(* PLC project pj23SH01.project, CODESYS CODESYS V3.5 SP18 Patch 2 *)
(* stored: creationDateTime 2023-05-12T09:11:09.1774968, modificationDateTime 2023-05-12T09:10:59.1943593 *)

TYPE EASY_object_manager_struct_t : STRUCT
  xFlip : BOOL;  (* commands *)
  xLoaded : BOOL;  (* feedbacks *)
  MarkerPose : ROS_pose_struct_t;
  xMarkerDetected : BOOL;
  xIsFlipped : BOOL;
  xResult_OK : BOOL;  (* elaboration *)
  xResult_NOT_OK : BOOL;
END_STRUCT;
END_TYPE

{attribute 'qualified_only'}
{attribute 'strict'}
TYPE piece_state_enum_t : (PieceUnknownState, PieceOK, PieceNotOK) UDINT;
END_TYPE

{attribute 'qualified_only'}
{attribute 'strict'}
TYPE manipulator_state_enum_t : (ManipulatorUnknownState, ManipulatorReady, ManipulatorRunning, ManipulatorError) UDINT;
END_TYPE

{attribute 'qualified_only'}
{attribute 'strict'}
TYPE piece_error_enum_t : (PIECE_NO_ERROR, PIECE_IN_WRONG_CONFIG, PIECE_NOT_FOUND) UDINT;
END_TYPE

{attribute 'qualified_only'}
{attribute 'strict'}
TYPE manipulator_error_enum_t : (MANIP_NO_ERROR, MANIP_GENERAL_ERROR, MANIP_EM_STOP, MANIP_EXEC_FAILED) UDINT;
END_TYPE

TYPE full_machine_struct_t : STRUCT
  Machine : machine_struct_t;
  Details : machine_details_struct_t;
  Counters : counters_interface_struct_t;
END_STRUCT;
END_TYPE

TYPE piece_struct_t : STRUCT
  xEnable : BOOL;
  eState : piece_state_enum_t;
  eError : piece_error_enum_t;
END_STRUCT;
END_TYPE

TYPE machine_struct_t : STRUCT
  xEnable : BOOL;
  eState : machine_state_enum_t;
  eError : machine_error_enum_t;
  sErrorMessage : STRING(255);
END_STRUCT;
END_TYPE

TYPE machine_details_struct_t : STRUCT
  aPieces : ARRAY[0..1] OF piece_struct_t;
  Manipulator : manipulator_struct_t;
END_STRUCT;
END_TYPE

TYPE manipulator_struct_t : STRUCT
  xEnable : BOOL;
  eState : manipulator_state_enum_t;
  eError : manipulator_error_enum_t;
END_STRUCT;
END_TYPE

TYPE counters_struct_t : STRUCT
  udiPiecesOK_Counter : UDINT;
  udiPiecesNotOK_Counter : UDINT;
  dtUTCStartCounting : DT;  (* time *)
  dwUpTime : DWORD;  (* in seconds *)
  dwReadyTime : DWORD;
  dwRunningTime : DWORD;  (* in seconds *)
  dwErrorTime : DWORD;  (* in seconds *)
END_STRUCT;
END_TYPE

TYPE counters_interface_struct_t : STRUCT
  LastSession : counters_struct_t;
  Overall : counters_struct_t;
END_STRUCT;
END_TYPE

TYPE ros_interface_struct_t_OLD : STRUCT
  xRun : BOOL;
  xRobotIsRunning : BOOL;
  diProcessCode : DINT;
  eProcessState : process_code_enum_t;
  sObjectCode : STRING;
END_STRUCT;
END_TYPE

TYPE light_tower_struct_t : STRUCT
  xGreen : BOOL;
  xYellow : BOOL;
  xRed : BOOL;
  xBuzzer : BOOL;
END_STRUCT;
END_TYPE

{attribute 'pack_mode' := '0'}
TYPE ROS_pose_struct_t : STRUCT
  position : ROS_position_struct_t;
  orientation : ROS_orientation_struct_t;
END_STRUCT;
END_TYPE

TYPE ROS_position_struct_t : STRUCT
  x : LREAL;
  y : LREAL;
  z : LREAL;
END_STRUCT;
END_TYPE

TYPE ROS_orientation_struct_t : STRUCT
  x : LREAL;
  y : LREAL;
  z : LREAL;
  w : LREAL;
END_STRUCT;
END_TYPE

TYPE ROS_ori_eu_struct_t : STRUCT
  lrRoll : LREAL;
  lrPitch : LREAL;
  lrYaw : LREAL;
END_STRUCT;
END_TYPE

TYPE ROS_pose_eu_struct_t : STRUCT
  position : ROS_pos_struct_t;
  orientation : ROS_ori_eu_struct_t;
  xIsValid : BOOL;
END_STRUCT;
END_TYPE

TYPE ROS_pos_struct_t : STRUCT
  lrX : LREAL;
  lrY : LREAL;
  lrZ : LREAL;
END_STRUCT;
END_TYPE

{attribute 'qualified_only'}
{attribute 'strict'}
TYPE eActionDoosan_t : (action_null := 0, action_go_to_carpos := 10, action_go_home := 1000) DINT;
END_TYPE

{attribute 'qualified_only'}
{attribute 'strict'}
TYPE eDoosanError_t : (error_ok := 0, error_invalid_input := 1, error_no_action := 2);
END_TYPE

TYPE doosan_t : STRUCT
  Joints : joints_t;
  Cartesian : cartesian_t;
  InfoRobot : info_robot_t;
  xIsAlive : BOOL;  (* 20/10/2022 *)
END_STRUCT;
END_TYPE

TYPE joints_t : STRUCT
  j1 : REAL;
  j2 : REAL;
  j3 : REAL;
  j4 : REAL;
  j5 : REAL;
  j6 : REAL;
END_STRUCT;
END_TYPE

TYPE cartesian_t : STRUCT
  x : REAL;
  y : REAL;
  z : REAL;
  A : REAL;
  B : REAL;
  C : REAL;
END_STRUCT;
END_TYPE

TYPE joint_temperature_t : STRUCT
  Temp_J1 : REAL;
  Temp_J2 : REAL;
  Temp_J3 : REAL;
  Temp_J4 : REAL;
  Temp_J5 : REAL;
  Temp_J6 : REAL;
END_STRUCT;
END_TYPE

TYPE joint_torque_t : STRUCT
  Torque_J1 : REAL;
  Torque_J2 : REAL;
  Torque_J3 : REAL;
  Torque_J4 : REAL;
  Torque_J5 : REAL;
  Torque_J6 : REAL;
END_STRUCT;
END_TYPE

TYPE info_robot_t : STRUCT
  temp_joints : joint_temperature_t;
  torque_joints : joint_torque_t;
END_STRUCT;
END_TYPE

TYPE zones_t : STRUCT
  a_iMoveX : INT;
  a_iMoveY : INT;
  a_iSaveCurrentPosX : INT;
  a_iSaveCurrentPosY : INT;
  a_iWight : INT;  (* - *)
  a_iHeight : INT;
  a_sPositionRectangle : STRING(20);  (* - *)
  a_xEnableMove : BOOL;  (* - *)
  a_xEnableBlocks : BOOL;  (* - *)
END_STRUCT;
END_TYPE

TYPE confzones_t : STRUCT
  zones_tractor : ARRAY[0..prg_Hmi_ZoneTractor.c_iMaxZone] OF zones_t;
END_STRUCT;
END_TYPE

TYPE dososa_responce_t : STRUCT
  xBusy : BOOL;
  xDone : BOOL;
  xError : BOOL;
  xAborted : BOOL;
  eErrorID : eDoosanError_t;
END_STRUCT;
END_TYPE

TYPE doosan_state_struct_t : STRUCT
  eRobotState : doosan_robot_state_enum_t;
  xSO_ServoOn : BOOL;
  xSS_SafetyStopped : BOOL;
  xES_EmergencyStopped : BOOL;
  xDTPB_DirectTeachButtonPressed : BOOL;
  xPBP_PowerButtonPressed : BOOL;
END_STRUCT;
END_TYPE

TYPE INCAS_box_info_struct_t : STRUCT
  time_stamp : STRING;
  box_code : STRING;
  batch_code : STRING;
  hub_code : STRING;
  palletizing_code : STRING;
  box_state : INT;
  dim_code : STRING;
  weight : STRING;
END_STRUCT;
END_TYPE

TYPE INCAS_box_ack_struct_t : STRUCT
  time_stamp : STRING;
  last_box_code : STRING;
  error_id : INT;
END_STRUCT;
END_TYPE

TYPE SysD_log_entry_t : STRUCT
  eSeverity : SysD_log_entry_severity_enum_t;
  sTimeStamp : STRING;
  sDescription : STRING(255);
  sComponent : STRING;
END_STRUCT;
END_TYPE

TYPE SysD_log_row_t : STRUCT
  diID : DINT;
END_STRUCT;
END_TYPE

TYPE db_t_items_struct_t : STRUCT
  sBoxCode : STRING;
  sBatchCode : STRING;
  sHubCode : STRING;
  sPalletizingCode : STRING;
  sDimCode : STRING;
  sInsertedAt : STRING;
END_STRUCT;
END_TYPE

TYPE test_ros_struct_t : STRUCT
  iInt : INT;
  rReal : REAL;
  lrLReal : LREAL;
  udiUdint : UDINT;
END_STRUCT;
END_TYPE

TYPE mission_list_elem_struct_t : STRUCT
  sTimestamp : STRING;
  sMissionID : STRING;
  sItemCode : STRING;
  sOrigin : STRING;
  sDestination : STRING;
END_STRUCT;
END_TYPE

TYPE mission_proc_elem_struct_t : STRUCT
  eProcessState : mission_process_state_enum_t;
  eProcessError : mission_process_error_enum_t;
END_STRUCT;
END_TYPE

TYPE buffer_struct_t : STRUCT
  Piston : SysD_CommonDevices.bistable_piston_struct_t;
  Inverter : SysD_CommonDevices.inverter_struct_t;
  axPositionSensors : ARRAY[0..GVL_Consts.gc_uiMaxIndBuffer] OF BOOL;
END_STRUCT;
END_TYPE

TYPE conveyor_struct_t : STRUCT
  aInverters : ARRAY[0..GVL_Consts.gc_uiMaxIndConveyorInverters] OF SysD_CommonDevices.inverter_struct_t;
  aLocations : ARRAY[0..GVL_Consts.gc_uiMaxIndConveyor] OF conveyor_loc_struct_t;
END_STRUCT;
END_TYPE

TYPE conveyor_loc_struct_t : STRUCT
  xPresenceSensorValue : BOOL;
  iBufferIndex : INT := GVL_Consts.gc_iDefault_UnassignedBufferIndex;
  Barrier : SysD_CommonDevices.bistable_piston_struct_t;
  xHasBarrier : BOOL;
  iInverterIndex : INT := GVL_Consts.gc_iDefault_UnassignedInverterIndex;
END_STRUCT;
END_TYPE

TYPE items_struct_t : STRUCT
  sItemCode : STRING;
  eLocationType : location_type_enum_t;  (* buffer? conveyor? *)
  iLocationIndex : INT;  (* e.g.: buffer ind 2, or e.g.: conveyor location 8 *)
  iLocationSubIndex : INT;  (* e.g.: buffer subindex 1, e.g. conveyor has no subindex, will be ignored (better set to "unassigned" constant) *)
  sMissionID : STRING;
END_STRUCT;
END_TYPE

TYPE db_t_commands_struct_t : STRUCT
  diID : DINT;
  sSourcePosition : STRING;
  sDestinationPosition : STRING;
  iCommandStatus : INT;
  sInserted : STRING;
  sUpdated : STRING;
END_STRUCT;
END_TYPE

TYPE PalletizingOptions : STRUCT
  tool_name : STRING;  (* Tool *)
  object_name : STRING;  (* Object *)
  object_weight : LREAL;
  pattern_file : STRING(255);  (* Pattern manager *)
  transform_name : STRING;
END_STRUCT;
END_TYPE

TYPE pallcube_pub_struct_t : STRUCT
  run : BOOL;
  lft_palletizing_options : PalletizingOptions;
  rgt_palletizing_options : PalletizingOptions;
  lifter_controller_feedback : CommonFeedback;
  lifter_controller_joint_states : JointState;
END_STRUCT;
END_TYPE

TYPE CommonCommand : STRUCT
  execute : BOOL;
  abort : BOOL;
  id : DINT;
END_STRUCT;
END_TYPE

TYPE CommonFeedback : STRUCT
  busy : BOOL;
  done : BOOL;
  aborted : BOOL;
  error : BOOL;
  error_id : DINT;
END_STRUCT;
END_TYPE

TYPE pallcube_sub_struct_t : STRUCT
  process_code : DINT;  (* Process *)
  is_running : BOOL;
  lifter_controller_command : CommonCommand;  (* Lifter *)
END_STRUCT;
END_TYPE

TYPE JointState : STRUCT
  header : Header_;
  {attribute 'robin_var_len'}
  name : ARRAY[1..Robin.DEF_ARRAY_LEN] OF STRING;
  {attribute 'robin_var_len'}
  position : ARRAY[1..Robin.DEF_ARRAY_LEN] OF LREAL;
  {attribute 'robin_var_len'}
  velocity : ARRAY[1..Robin.DEF_ARRAY_LEN] OF LREAL;
  {attribute 'robin_var_len'}
  effort : ARRAY[1..Robin.DEF_ARRAY_LEN] OF LREAL;
END_STRUCT;
END_TYPE

TYPE ros_to_codesys_struct_t : STRUCT
  Subscripted : pallcube_sub_struct_t;
  eProcessState : process_code_enum_t;
END_STRUCT;
END_TYPE

TYPE codesys_to_ros_struct_t : STRUCT
  Published : pallcube_pub_struct_t;
END_STRUCT;
END_TYPE

TYPE ros_interface_struct_t : STRUCT
  Codesys2ROS : codesys_to_ros_struct_t;
  ROS2Codesys : ros_to_codesys_struct_t;
END_STRUCT;
END_TYPE

TYPE Header_ : STRUCT
  seq : UDINT;
  stamp : ROS_TIME;
  frame_id : STRING(83);
END_STRUCT;
END_TYPE

TYPE TestStruct : STRUCT
  var_bool : BOOL;
  var_byte : BYTE;
  var_int16 : INT;
  var_uint64 : ULINT;
  var_float32 : REAL;
  var_float64 : LREAL;
  var_string : STRING;
  var_pose : Pose;
  var_struct_array : ARRAY[1..2] OF ByteMultiArray;
  {attribute 'robin_var_len'}
  var_struct_varlen_array : ARRAY[1..2] OF ByteMultiArray;
END_STRUCT;
END_TYPE

{attribute 'qualified_only'}
{attribute 'strict'}
TYPE e_main_pages_t : (home := 0, error_frame := 1, application := 2, mini_pc := 3, interface_settings := 4);
END_TYPE

{attribute 'qualified_only'}
{attribute 'strict'}
TYPE e_main_minipcmenu_t : (menu := 0, minipc_manager := 1);
END_TYPE

(* values of e_page_robot_t: sorters: compose_pallet:=5, *)

{attribute 'qualified_only'}
{attribute 'strict'}
TYPE e_page_robot_t : (menu := 0, application := 1, manipulator_converter := 2, config_pallet := 3, opcua_tests := 4, sorters := 5);
END_TYPE

TYPE confzones_t : STRUCT
  zones_tractor : ARRAY[0..prg_Hmi_ZoneTractor.c_iMaxZone] OF zones_t;
END_STRUCT;
END_TYPE

TYPE zones_t : STRUCT
  a_iMoveX : INT;
  a_iMoveY : INT;
  a_iSaveCurrentPosX : INT;
  a_iSaveCurrentPosY : INT;
  a_iWight : INT;  (* - *)
  a_iHeight : INT;
  a_sPositionRectangle : STRING(20);  (* - *)
  a_xEnableMove : BOOL;  (* - *)
  a_xEnableBlocks : BOOL;  (* - *)
END_STRUCT;
END_TYPE

TYPE synoptic_boxes_info_struct_t : STRUCT
  sBoxCode : STRING;
  xInvisible : BOOL;
END_STRUCT;
END_TYPE

TYPE mapping_info_struct_t : STRUCT
  sLocationName : STRING;
  eType : sorter_elem_type_enum_t;
  Info : sorter_elem_info_union_t;
END_STRUCT;
END_TYPE

TYPE buffer_elem_info_struct_t : STRUCT
  iSectionIndex : INT;
  iNumber : INT;
  iDepth : INT;
END_STRUCT;
END_TYPE

TYPE conveyor_elem_info_struct_t : STRUCT
  iLocationIndex : INT;
END_STRUCT;
END_TYPE

TYPE sorter_elem_info_union_t : UNION
  BufferInfo : buffer_elem_info_struct_t;
  ConveyorInfo : conveyor_elem_info_struct_t;
END_UNION;
END_TYPE

{attribute 'qualified_only'}
VAR_GLOBAL CONSTANT  (* GVL *)
  c_MaxConfings : INT := 1;
END_VAR

{attribute 'qualified_only'}
VAR_GLOBAL CONSTANT  (* GVL_Consts *)
  gc_uiBufferDepth : UINT := 5;  (* buffers *)
  gc_uiMaxIndBuffer : UINT := (gc_uiBufferDepth - 1);
  gc_uiConveyorLocations : UINT := (ANY_TO_UINT(gc_iMaxIndBuffers) + 2);  (* conveyor *)
  gc_uiMaxIndConveyor : UINT := (gc_uiConveyorLocations - 1);
  gc_uiConveyorInvertersNum : UINT := gc_uiConveyorLocations;
  gc_uiMaxIndConveyorInverters : UINT := (gc_uiConveyorInvertersNum - 1);
  gc_iMaxIndInput : INT := 30;  (* input/output interface *)
  gc_iMaxIndOutput : INT := 30;
  gc_iMaxIndBuffers : INT := 15;
  gc_iItemsNum : UINT := 50;  (* items *)
  gc_iMaxIndItems : UINT := (gc_iItemsNum - 1);
  gc_iDefault_UnassignedInverterIndex : INT := -1;  (* default values *)
  gc_iDefault_UnassignedBufferIndex : INT := -1;
  gc_iDefault_UnassignedLocationIndex : INT := -1;
END_VAR

{attribute 'qualified_only'}
VAR_GLOBAL CONSTANT  (* GVL_ROSConsts *)
  c_uiJointStateNum : UINT := 1;
  c_uiMaxIndJointState : UINT := c_uiJointStateNum;
END_VAR

INTERFACE ILogEntry
PROPERTY LogEntry : SysD_log_entry_t
END_PROPERTY
END_INTERFACE

INTERFACE ITF_Sorter
METHOD METH_Map : INT
END_METHOD
END_INTERFACE

FUNCTION FUN_DB_insert_log_entry : SysD_DB.SysD_MySQLQuery
  VAR_INPUT
    SysD_LogEntry : SysD_log_entry_t;
  END_VAR
  VAR_OUTPUT
    diLength : DINT;
    xWarningLongQuery : BOOL;
  END_VAR
  VAR
    sRes : STRING(500);  (* sRes : SysD_DB.SysD_MySQLQuery; *)
    iBufferSize : INT;
    sAux : STRING(255);
    sTypeOfRequest : STRING;
    diMaxLength : DINT;
  END_VAR

            iBufferSize := __UXINT_TO_INT(XSIZEOF(sRes));

// procedure
STU.StrConcatA(pstTo := ADR(sRes), pstFrom := ADR('insert into t_log(severity, time_stamp, description, component) values ('), iBufferSize := iBufferSize);

// severity
SysMem.SysMemSet(pDest := ADR(sAux), udiCount := XSIZEOF(sAux), udiValue := 0);
sAux := TO_STRING(SysD_LogEntry.eSeverity);
STU.StrConcatA(pstTo := ADR(sRes), pstFrom := ADR(sAux), iBufferSize := iBufferSize);

STU.StrConcatA(pstTo := ADR(sRes), pstFrom := ADR(', '), iBufferSize := iBufferSize); // separator

// time stamp
SysMem.SysMemSet(pDest := ADR(sAux), udiCount := XSIZEOF(sAux), udiValue := 0);
sAux := SysD_DB.FUN_ConvertToSQLQueryString(sString := SysD_LogEntry.sTimeStamp);
STU.StrConcatA(pstTo := ADR(sRes), pstFrom := ADR(sAux), iBufferSize := iBufferSize);

STU.StrConcatA(pstTo := ADR(sRes), pstFrom := ADR(', '), iBufferSize := iBufferSize); //separator

// description
SysMem.SysMemSet(pDest := ADR(sAux), udiCount := XSIZEOF(sAux), udiValue := 0);
sAux := SysD_DB.FUN_ConvertToSQLQueryString(sString := SysD_LogEntry.sDescription);
STU.StrConcatA(pstTo := ADR(sRes), pstFrom := ADR(sAux), iBufferSize := iBufferSize);

STU.StrConcatA(pstTo := ADR(sRes), pstFrom := ADR(', '), iBufferSize := iBufferSize); //separator

// component
SysMem.SysMemSet(pDest := ADR(sAux), udiCount := XSIZEOF(sAux), udiValue := 0);
sAux := SysD_DB.FUN_ConvertToSQLQueryString(sString := SysD_LogEntry.sComponent);
STU.StrConcatA(pstTo := ADR(sRes), pstFrom := ADR(sAux), iBufferSize := iBufferSize);

STU.StrConcatA(pstTo := ADR(sRes), pstFrom := ADR(');'), iBufferSize := iBufferSize); // terminator

diLength := STU.StrLenA(pstData := ADR(sRes));
diMaxLength := TO_DINT(XSIZEOF(SysD_DB.SysD_MySQLQuery)) - 1;
xWarningLongQuery := diLength > diMaxLength;
	

FUN_DB_insert_log_entry := sRes;


          
END_FUNCTION

FUNCTION FUN_GetLocalRTCString : STRING
  VAR
    dwRTC : DWORD;
    RTS_RTCRes : RTS_IEC_RESULT;
    dtRTCTime : DT;
    sRTCTime : STRING;
    udiResUTCLocal : RTS_IEC_RESULT;
    dwRTC_Local : DWORD;
    udiHighRes : RTS_IEC_RESULT;
    uliHighResTimestamp : SYSTIME;
    dwMilliSec : DWORD;
    sAux : STRING(255);
  END_VAR

            // dwRTC := SysTimeRtc.SysTimeRtcGet(pResult := RTS_RTCRes);
udiHighRes := SysTimeRtc.SysTimeRtcHighResGet(pTimestamp := uliHighResTimestamp);
dwMilliSec := TO_DWORD(uliHighResTimestamp MOD 1000);//02/11/2022
sAux := TO_STRING(dwMilliSec);
IF dwMilliSec < 10 THEN
	sAux := CONCAT('00', sAux);
ELSIF dwMilliSec < 100 THEN
	sAux := CONCAT('0', sAux);
END_IF
dwRTC := TO_DWORD(uliHighResTimestamp / 1000);
udiResUTCLocal := SysTimeRTCConvertUTCToLocal(dwTimestampUtc := dwRTC, pdwTimestampLocal := dwRTC_Local);
dtRTCTime := DWORD_TO_DT(dwRTC_Local);
sRTCTime := DT_TO_STRING(dtRTCTime);
sRTCTime := CONCAT(sRTCTime, '.');
sRTCTime := CONCAT(sRTCTime, sAux);

FUN_GetLocalRTCString := sRTCTime;
          
END_FUNCTION

(* returns 0 if parameters are ok *)
FUNCTION FUN_AddToALogEntryQueue : INT
  VAR_INPUT
    LogEntry : SysD_log_entry_t;
    pdiCounter : POINTER TO DINT := 0;
  END_VAR
  VAR_IN_OUT
    itfQueueOfLogEntries : COL.Queue;
  END_VAR
  VAR_OUTPUT
    xFullBuffer : BOOL;
    eColError : COL.COLLECTION_ERROR;
  END_VAR
  VAR
    eColRes : COL.COLLECTION_ERROR;
    LogEntriesFactory : LogEntryElementFactory;
    eLogEntryFactErr : FBF.ERROR;
    iRes : INT;
    udiNumElement : UDINT;
  END_VAR

            LogEntry.sTimeStamp := FUN_GetLocalRTCString();

eColRes := itfQueueOfLogEntries.AddElement(
	itfElement := LogEntriesFactory.Create(
		Value := LogEntry, 
		eError => eLogEntryFactErr
	)
);
IF eColRes = COL.COLLECTION_ERROR.NO_ERROR THEN
// 	diCounter := (diCounter + 1) MOD 16#7FFFFFFF;
	IF pdiCounter > 0 THEN //increment counter if passed as pointer
		pdiCounter^ := (pdiCounter^ + 1) MOD 16#7FFFFFFF;
	END_IF
ELSE
	xFullBuffer := eColRes = COL.COLLECTION_ERROR.MAXIMUM_SIZE_OF_ELEMENTS_EXCEEDED;
END_IF

udiNumElement := itfQueueOfLogEntries.CountElements(); // debugging purposes

eColError := eColRes;
FUN_AddToALogEntryQueue := iRes;
          
END_FUNCTION

(* returns 0 if parameters are ok *)
FUNCTION FUN_PollFromALogEntryQueue : INT
  VAR_INPUT
    pdiCounter : POINTER TO DINT := 0;
  END_VAR
  VAR_IN_OUT
    itfQueueOfLogEntries : COL.Queue;
  END_VAR
  VAR_OUTPUT
    LogEntry : SysD_log_entry_t;
    eColError : COL.COLLECTION_ERROR;
  END_VAR
  VAR
    itfQueue : COL.IQueue2;
    eColRes : COL.COLLECTION_ERROR;
    itfCOLElement : COL.IElement;
    itfLogEntryElement : ILogEntry;
    xCompatibleItf : BOOL;
    iRes : INT;
    xResult : BOOL;
  END_VAR

            xResult := __QUERYINTERFACE(itfQueueOfLogEntries, itfQueue);
IF xResult THEN
	eColRes := itfQueueOfLogEntries.Poll(itfElement => itfCOLElement);
	xCompatibleItf := __QUERYINTERFACE(itfCOLElement, itfLogEntryElement);
	IF xCompatibleItf THEN
		LogEntry := itfLogEntryElement.LogEntry;
		pdiCounter^ := (pdiCounter^ + 1) MOD 16#7FFFFFFF;
	ELSE
		iRes := -2;
	END_IF
ELSE
	iRes := -1;
END_IF

eColError := eColRes;
FUN_PollFromALogEntryQueue := iRes;
          
END_FUNCTION

FUNCTION_BLOCK SQL_Interp_GetLog EXTENDS SysD_DB.SQL_QueryInterpr_TPL

            
          

(* {warning 'Add method implementation '} *)
METHOD METH_GetNewKey : BOOL
  VAR_INPUT
    iInd : INT;
  END_VAR
  VAR_OUTPUT
    xwSize : __XWORD;
  END_VAR
  VAR
    pDestStruct : POINTER TO SysD_log_row_t;
    xRes : BOOL;
  END_VAR
                  pDestStruct := pSpecDestStruct;
CASE iInd OF
	0:
		sKey := 'id';
		pStartColumn := ADR(pDestStruct^.diID);
		VAR_INFO_ThisCol := __VARINFO(pDestStruct^.diID);
	1:
		sKey := 'severity';
		pStartColumn := ADR(pDestStruct^.eSeverity);
		VAR_INFO_ThisCol := __VARINFO(pDestStruct^.eSeverity);
	2:
		sKey := 'time_stamp';
		pStartColumn := ADR(pDestStruct^.sTimeStamp);
		VAR_INFO_ThisCol := __VARINFO(pDestStruct^.sTimeStamp);
	3:
		sKey := 'description';
		pStartColumn := ADR(pDestStruct^.sDescription);
		VAR_INFO_ThisCol := __VARINFO(pDestStruct^.sDescription);
	4:
		sKey := 'component';
		pStartColumn := ADR(pDestStruct^.sComponent);
		VAR_INFO_ThisCol := __VARINFO(pDestStruct^.sComponent);
	5:
		xRes := TRUE;
END_CASE

xwSize := XSIZEOF(pDestStruct^); // must


METH_GetNewKey := xRes;
                
END_METHOD
END_FUNCTION_BLOCK

{attribute 'enable_dynamic_creation'}
{attribute 'hide'}
FUNCTION_BLOCK LogEntryData EXTENDS FBF.InstanceData
  VAR_INPUT
    LogEntry : SysD_log_entry_t;
  END_VAR

            (* !! Do not add any executable code here !! *)
SUPER^();
          
END_FUNCTION_BLOCK

(* Demo element with two integer values. An element must implement an interface which extends |COL.IElement|. This function block extends FBF.InstanceBase to enable dynamic creation via FBFactory. *)
{attribute 'no_explicit_call' := 'Explicit calls not allowed.'}
FUNCTION_BLOCK LogEntryElement EXTENDS FBF.InstanceBase IMPLEMENTS ILogEntry
  VAR_INPUT
    {attribute 'input_constant'}
    LogEntryValue : SysD_log_entry_t;
  END_VAR

            
          

(* Returns true of this element and itfElement are equal. This method will be called from the function block |COL.HashTable| to find an element by key if the hashcode of an element collides with an other element. IMPORTANT: The underlying value to be compared with MUST NOT be changed during the lifecycle of the object. *)
METHOD ElementEquals : BOOL
  VAR_INPUT
    itfElement : COL.IElement;  (* The element to compare *)
  END_VAR
  VAR
    itfLogEntryElement : ILogEntry;
    Aux : SysD_log_entry_t;
    Aux2 : SysD_log_entry_t;
    xResult : BOOL;
  END_VAR
                  xResult := __QUERYINTERFACE(itfElement, itfLogEntryElement);
IF xResult THEN
	Aux := LogEntryValue;
	Aux2 := itfLogEntryElement.LogEntry;
	ElementEquals := Aux.sTimeStamp = Aux2.sTimeStamp;	
ELSE
	ElementEquals := FALSE;
END_IF 
                
END_METHOD

(* Returns the hashcode of this element. This method is used by hash based collections (e.g. |Hashtable|) to get the hashcode from a element. IMPORTANT: The value of the method MUST NOT be changed during the lifecycle of the object. *)
METHOD ElementHashCode : LINT
                  // ElementHashCode := TO_LINT(sValue);
ElementHashCode := TO_LINT(LogEntryValue.sTimeStamp);

                
END_METHOD

(* Compares this element with itfElement. Returns 0 if the elements are equal, < 0 if the element is less than itfElement, > 0 if the element is greater than itfElement. This method will be called from sorted collections (e.g. |COL.SortedList|) to sort the elements. IMPORTANT: The underlying value to be compared with MUST NOT be changed during the lifecycle of the object. *)
METHOD ElementCompareTo : INT
  VAR_INPUT
    itfElement : COL.IElement;  (* The element to compare *)
  END_VAR
  VAR
    itfLogEntryElement : ILogEntry;
    Aux : SysD_log_entry_t;
    Aux2 : SysD_log_entry_t;
    xResult : BOOL;
    uliTimestamp1 : ULINT;
    uliTimestamp2 : ULINT;
  END_VAR
                  // We use integer iInt1 for sorting.
xResult := __QUERYINTERFACE(itfElement, itfLogEntryElement);
IF xResult THEN
	Aux := itfLogEntryElement.LogEntry;
	Aux2 := LogEntryValue;
	uliTimestamp1 := DT_TO_ULINT(STRING_TO_DT(Aux.sTimeStamp));
	uliTimestamp2 := DT_TO_ULINT(STRING_TO_DT(Aux2.sTimeStamp));
	IF uliTimestamp2 < uliTimestamp1 THEN
		ElementCompareTo := -1;
	ELSIF uliTimestamp2 > uliTimestamp1 THEN
		ElementCompareTo := 1;
	ELSE
		ElementCompareTo := 0;
	END_IF
ELSE
	ElementCompareTo := -1;
END_IF 

                
END_METHOD

(* This methode is called from the factory to give a chance to initialize the new fb instance with the content of itfData *)
METHOD prvInstInit : FBF.ERROR
  VAR_INPUT
    itfData : FBF.IData;
  END_VAR
  VAR
    pData : POINTER TO LogEntryData;
    xOk : BOOL;
  END_VAR
                  SUPER^.prvInstInit(itfData);
xOk := __QUERYPOINTER(itfData, pData);
IF xOk THEN
	THIS^.LogEntry := pData^.LogEntry;
END_IF

                
END_METHOD

PROPERTY LogEntry : SysD_log_entry_t
GET
                    LogEntry := LogEntryValue;
                  
END_GET
SET
                    LogEntryValue := LogEntry;
                  
END_SET
END_PROPERTY
END_FUNCTION_BLOCK

{attribute 'enable_dynamic_creation'}
FUNCTION_BLOCK LogEntryElementFactory EXTENDS FBF.FactoryBase

            SUPER^();

          

(* Creates a IntElement *)
METHOD Create : ILogEntry
  VAR_INPUT
    Value : SysD_log_entry_t;
  END_VAR
  VAR_OUTPUT
    eError : FBF.ERROR;
  END_VAR
  VAR
    hInst : CAA.HANDLE;
    itfInst : FBF.IInstance;
    xOk : BOOL;
    itfData : LogEntryData;
    pInstance : POINTER TO LogEntryElement;
  END_VAR
                  (* !!! This code must not be subject to change !!! *)
itfData(LogEntry:=Value);
hInst := SUPER^.prvAllocInstMem(eError => eError);
pInstance := SUPER^.prvGetInstPointer(hInst);
IF pInstance <> 0 AND eError = FBF.ERROR.NO_ERROR THEN

	{implicit on}
	pInstance^.__vfInit();
	pInstance^.FB_Init(TRUE, FALSE);
	{implicit off}

	xOk := __QUERYINTERFACE(pInstance^, itfInst);
	IF xOk THEN
		xOk := SUPER^.prvInstInit(itfInst, hInst, itfData, eError=>eError);
	ELSE
		eError := FBF.ERROR.WRONG_INTERFACE;
	END_IF

	IF NOT xOk THEN
		SUPER^.prvFreeInstMem(hInst);
		Create := CAA.gc_pNULL;
    ELSE
        __QUERYINTERFACE(pInstance^, Create);
	END_IF
END_IF

                
END_METHOD

(* {attribute 'conditionalshow' := 'SomeText'} {attribute 'conditionalshow'} {attribute 'hide'} *)
PROPERTY prvInstCount : CAA.COUNT
GET
                    (* Please choose a proper value for prvInstCount *)
prvInstCount := 100;
                  
END_GET
END_PROPERTY

(* {attribute 'conditionalshow' := 'SomeText'} {attribute 'conditionalshow'} {attribute 'hide'} *)
PROPERTY prvInstPoolExtendsFactor : USINT
GET
                    (* Please choose a proper value for prvInstPoolExtendsFactor *)
(* This value will be interpreted as a 0..x% size extendsion related to the original size of the pool *)
prvInstPoolExtendsFactor := 50; //20
                  
END_GET
END_PROPERTY

(* {attribute 'conditionalshow' := 'SomeText'} {attribute 'conditionalshow'} {attribute 'hide'} *)
PROPERTY prvInstSize : CAA.SIZE
GET
                    (* Please replace CustomFB with your specific function block type *)
prvInstSize := XSIZEOF(LogEntryElement);
                  
END_GET
END_PROPERTY
END_FUNCTION_BLOCK

FUNCTION_BLOCK SQL_Interp_GetItems EXTENDS SysD_DB.SQL_QueryInterpr_TPL

            
          

(* {warning 'Add method implementation '} *)
METHOD METH_GetNewKey : BOOL
  VAR_INPUT
    iInd : INT;
  END_VAR
  VAR_OUTPUT
    xwSize : __XWORD;
  END_VAR
  VAR
    pDestStruct : POINTER TO db_t_items_struct_t;
    xRes : BOOL;
  END_VAR
                  pDestStruct := pSpecDestStruct;
CASE iInd OF
	0:
		sKey := 'box_code';
		pStartColumn := ADR(pDestStruct^.sBoxCode);
		VAR_INFO_ThisCol := __VARINFO(pDestStruct^.sBoxCode);
	1:
		sKey := 'batch_code';
		pStartColumn := ADR(pDestStruct^.sBatchCode);
		VAR_INFO_ThisCol := __VARINFO(pDestStruct^.sBatchCode);
	2:
		sKey := 'hub_code';
		pStartColumn := ADR(pDestStruct^.sHubCode);
		VAR_INFO_ThisCol := __VARINFO(pDestStruct^.sHubCode);
	3:
		sKey := 'palletizing_code';
		pStartColumn := ADR(pDestStruct^.sPalletizingCode);
		VAR_INFO_ThisCol := __VARINFO(pDestStruct^.sPalletizingCode);
	4:
		sKey := 'dim_code';
		pStartColumn := ADR(pDestStruct^.sDimCode);
		VAR_INFO_ThisCol := __VARINFO(pDestStruct^.sDimCode);
	5:
		sKey := 'inserted_at';
		pStartColumn := ADR(pDestStruct^.sInsertedAt);
		VAR_INFO_ThisCol := __VARINFO(pDestStruct^.sInsertedAt);
	6:
		xRes := TRUE;
END_CASE

xwSize := XSIZEOF(pDestStruct^); // must


METH_GetNewKey := xRes;
                
END_METHOD
END_FUNCTION_BLOCK

FUNCTION_BLOCK FB_Sorter_TPL EXTENDS CBML.LConC IMPLEMENTS ITF_Sorter
  VAR_INPUT
    aMissionsToDo : ARRAY[0..GVL_Consts.gc_iMaxIndInput] OF mission_list_elem_struct_t;
    iLastLocationIndex : INT;
  END_VAR
  VAR_OUTPUT
    aMissionProcessing : ARRAY[0..GVL_Consts.gc_iMaxIndOutput] OF mission_proc_elem_struct_t;
    uiErrorID : UINT;
  END_VAR
  VAR_IN_OUT
    aBuffers : ARRAY[0..GVL_Consts.gc_iMaxIndBuffers] OF buffer_struct_t;  (* input substructures are externally updated, output substructures directly set IOs *)
    Conveyor : conveyor_struct_t;  (* input substructures are externally updated, output substructures directly set IOs *)
  END_VAR
  VAR
    _iLastLocationIndex : INT := GVL_Consts.gc_iDefault_UnassignedLocationIndex;
    _aItemsStates : ARRAY[0..GVL_Consts.gc_iMaxIndItems] OF items_struct_t;
  END_VAR

            IF METH_IsValidLocationIndex(iIndex := iLastLocationIndex) THEN
	_iLastLocationIndex := iLastLocationIndex;
ELSE
	_iLastLocationIndex := TO_INT(XSIZEOF(Conveyor.aLocations)/XSIZEOF(Conveyor.aLocations[0])) - 1;
END_IF

SUPER^();
uiErrorID := TO_UINT(_Model.iErrorID);


(* CBLM actions *)
// SampleAction();
// StartAction();
// CyclicAction();
// CleanupAction();
// ResetAction();
          

ACTION ACT_HandleExternalContextWarning:
                IF NOT __ISVALIDREF(Conveyor) THEN
	RETURN;
END_IF

IF NOT __ISVALIDREF(aBuffers) THEN
	RETURN;
END_IF
              
END_ACTION

(* {warning 'Add method implementation '} ``CleanupAction`` is running until one of the following events occurs: When ``xComplete`` is ``TRUE`` the state |STATE.DONE| is reached. When ``xAbort`` is ``TRUE`` the state |STATE.ABORTED| is reached. When ``iErrorID`` ≠ 0 (Zero) the state |STATE.ERROR| is reached. | After a *Ready Condition* as input (``iErrorIDProposed`` = 0 and ``xAbortProposed`` = ``FALSE``), only the output states | `DONE` (``xComplete`` is ``TRUE``) or `ERROR` (``iErrorID`` ≠ 0) are possible. | After a *Error Condition* as input (``iErrorIDProposed`` ≠ 0), only the output state | `ERROR` (``iErrorID`` ≠ 0) is possible. | After a *Abort Condition* as Input (``xAbortProposed`` = ``TRUE``), only the output states | `ABORTED` (``xAbort`` is ``TRUE``) or `ERROR` (``iErrorID`` ≠ 0) are possible. .. admonition:: Example .. code-block:: codesys ( * common cleanup -- first steps * ) IF xComplete THEN IF xAbortProposed THEN ( * abort condition -- abort specific cleanup * ) xAbort := TRUE; xComplete := FALSE; ELSIF iErrorIDProposed <> 0 THEN ( * error condition -- error specific cleanup * ) iErrorID := SEL(xComplete, 0, iErrorIDProposed); xComplete := FALSE; ELSE ( * ready condition -- done specific cleanup* ) END_IF END_IF ( * common cleanup -- last steps * ) *)
METHOD CleanupAction
  VAR_INPUT
    xAbortProposed : BOOL;
    iErrorIDProposed : INT;
  END_VAR
  VAR_OUTPUT
    xComplete : BOOL;
    xAbort : BOOL;
    iErrorID : INT;
  END_VAR
                  IF xComplete THEN
	 IF xAbortProposed THEN
		 (* abort condition -- abort specific cleanup *)
		 xAbort := TRUE;
		 xComplete := FALSE;
	 ELSIF iErrorIDProposed <> 0 THEN
		 (* error condition -- error specific cleanup *)
		 iErrorID := SEL(xComplete, 0, iErrorIDProposed);
		 xComplete := FALSE;
	 ELSE
		(* ready condition -- done specific cleanup*)
		//sStatusMessage := 'Cleanup done';
     END_IF
END_IF
                
END_METHOD

(* The CyclicAction is running until either ``xComplete`` is ``TRUE`` or ``iErrorID`` ≠ 0 (Zero). If ``xComplete`` is ``TRUE`` or ``iErrorID`` ≠ 0 (Zero) the state |STATE.CLEANING| is reached. With ``itfTimingController`` ≠ 0 (Zero) it is possible to check the current invocation time (see: |ITimingController.ControllerCheckTiming|). Function blocks with a ``udiTimeLimit`` input variable (see: |IETrigTl|, |IETrigATl|, |IETrigTlTo|, |IETrigATlTo|, |ILConTl|, |ILConTlTo|, |ILConTlC|) should be implement in such a way that the current invocation is exited when the consumed time for this invocation has exceeded the settings from udiTimeLimit. .. admonition:: Example .. code-block:: codesys REPEAT // working to reach the ready condition // ⇒ xComplete := TRUE // if the maximum invocation time is reached // ⇒ xTimeLimit := TRUE // if the maximum operating time is reached // ⇒ xTimeOut := TRUE // if an error condition is reached // ⇒ set iErrorID to a value other than 0 (Zero) itfTimingController.ControllerCheckTiming( xTimeOut=>xTimeOut, xTimeLimit=>xTimeLimit ); xComplete := TRUE; iErrorID := ERROR.NO_ERROR; UNTIL xComplete OR xTimeOut OR xTimeLimit OR iErrorID <> ERROR.NO_ERROR END_REPEAT *)
METHOD CyclicAction
  VAR_INPUT
    itfTimingController : CBML.ITimingController;
  END_VAR
  VAR_OUTPUT
    xComplete : BOOL;
    iErrorID : INT;
  END_VAR
                  {warning disable C0371}
ACT_HandleExternalContextWarning();

// implementation

{warning enable C0371}

                
END_METHOD

(* This method is intended for releasing external resources (like RTS handles). Do not call other internal function block instances in the context of this method. Call only external functions defined inside the RTS. For cleaning up other resources then external ones, please use the ``CleanupAction``. This method should be callable in the context of ``FB_EXIT`` for example before downloading a new application or before reseting an application. *)
METHOD ExitAction
  VAR_INPUT
    xAfterCleanup : BOOL;
    xInCopyCode : BOOL;
  END_VAR
                  
                
END_METHOD

(* {warning 'Add method implementation '} The ``ResetAction`` is running until the output ``xComplete`` is ``TRUE``. If ``xComplete`` is ``TRUE`` the state |STATE.DORMANT| is reached. *)
METHOD ResetAction
  VAR_OUTPUT
    xComplete : BOOL;
  END_VAR
                  {message 'Complete method implementation '}
xComplete := TRUE;
                
END_METHOD

(* {warning 'Add method implementation '} The ``StartAction`` is running until either the output ``xComplete`` is ``TRUE`` or ``iErrorID`` ≠ 0 (Zero). If ``xComplete`` is ``TRUE`` the state |STATE.EXECUTING| is reached. If there is a ``iErrorID`` ≠ 0 (Zero) the state |STATE.CLEANING| is reached. .. note:: To sample the inputs in the first invocation of a function block the method SampleAction is the solution of choice. See: |ISampleActionProvider.SampleAction| *)
METHOD StartAction
  VAR_OUTPUT
    xComplete : BOOL;
    iErrorID : INT;
  END_VAR
                  {message 'Complete method implementation '}

IF METH_Check_UnassignedInverterIndexes() THEN
	iErrorID := TO_INT(sorter_error_enum_t.INCOMPLETE_MAPPING);
ELSE
	xComplete := TRUE;
END_IF

                
END_METHOD

METHOD METH_IsValidBufferIndex : BOOL
  VAR_INPUT
    iIndex : INT;
  END_VAR
  VAR
    iMaxIndex : INT;
  END_VAR
                  iMaxIndex := TO_INT(XSIZEOF(aBuffers)/XSIZEOF(aBuffers[0])) - 1;
METH_IsValidBufferIndex := iIndex >= 0 AND iIndex <= iMaxIndex;
                
END_METHOD

METHOD METH_IsValidInverterIndex : BOOL
  VAR_INPUT
    iIndex : INT;
  END_VAR
  VAR
    iMaxIndex : INT;
  END_VAR
                  iMaxIndex := TO_INT(XSIZEOF(Conveyor.aInverters)/XSIZEOF(Conveyor.aInverters[0])) - 1;
METH_IsValidInverterIndex := iIndex >= 0 AND iIndex <= iMaxIndex;
                
END_METHOD

METHOD METH_IsValidLocationIndex : BOOL
  VAR_INPUT
    iIndex : INT;
  END_VAR
  VAR
    iMaxIndex : INT;
  END_VAR
                  iMaxIndex := TO_INT(XSIZEOF(Conveyor.aLocations)/XSIZEOF(Conveyor.aLocations[0])) - 1;
METH_IsValidLocationIndex := iIndex >= 0 AND iIndex <= iMaxIndex;
                
END_METHOD

(* Useful? Must be cyclically invoked Copies value from first location of the mapped buffer to the conveyor *)
METHOD METH_GetConveyorSensorValuesFromBuffers : INT
  VAR
    iMaxInd : INT;
    iInd : INT;
    iBufferValue : INT;
    xIsValidBufferValue : BOOL;
    xValidMapping : BOOL;
    iCount : INT;
  END_VAR
                  {warning disable C0371}
ACT_HandleExternalContextWarning();

iMaxInd := TO_INT(XSIZEOF(Conveyor.aLocations)/XSIZEOF(Conveyor.aLocations[0])) - 1;
FOR iInd := 0 TO iMaxInd DO
	iBufferValue := Conveyor.aLocations[iInd].iBufferIndex;
	xIsValidBufferValue := METH_IsValidBufferIndex(iIndex := iBufferValue);
	
	xValidMapping := 
		xIsValidBufferValue
	; // AND ...
	IF xValidMapping THEN
		Conveyor.aLocations[iInd].xPresenceSensorValue := aBuffers[iBufferValue].axPositionSensors[0];
		iCount := iCount + 1;
	END_IF
END_FOR

METH_GetConveyorSensorValuesFromBuffers := iCount;

{warning enable C0371}
                
END_METHOD

METHOD METH_Check_UnassignedInverterIndexes : BOOL
  VAR
    iMaxInd : INT;
    iInd : INT;
    xUnassigned : BOOL;
    xRes : BOOL;
  END_VAR
                  {warning disable C0371}
ACT_HandleExternalContextWarning();

iMaxInd := TO_INT(XSIZEOF(Conveyor.aLocations)/XSIZEOF(Conveyor.aLocations[0])) - 1;
FOR iInd := 0 TO _iLastLocationIndex DO
	xUnassigned := Conveyor.aLocations[iInd].iInverterIndex = GVL_Consts.gc_iDefault_UnassignedInverterIndex;
	IF xUnassigned THEN
		xRes := TRUE;
		EXIT;
	END_IF
END_FOR

METH_Check_UnassignedInverterIndexes := xRes;

{warning enable C0371}
                
END_METHOD

(* Must be called at least once. This method maps the interchange locations to move items between the conveyor and one of the buffers *)
METHOD METH_Map : INT
                  {warning disable C0371}
ACT_HandleExternalContextWarning();
(*
Example:

Conveyor.aPositionSensors[1].iBufferIndex := 0; // shall be hard-coded depending on the physical implementation
Conveyor.aPositionSensors[2].iBufferIndex := 1; // shall be hard-coded depending on the physical implementation
...



*)

{warning enable C0371}

                
END_METHOD

METHOD METH_SetInverterLocationsRange : INT
  VAR_INPUT
    uiInverterIndex : UINT;
    uiFrom : UINT;
    uiTo : UINT;
  END_VAR
  VAR
    iMaxIndInverters : INT;
    xRangeValid : BOOL;
    xParsingOK : BOOL;
    iRes : INT;
    iInd : INT;
    xInverterIndexOK : BOOL;
  END_VAR
                  {warning disable C0371}
ACT_HandleExternalContextWarning();

iMaxIndInverters := TO_INT(XSIZEOF(Conveyor.aInverters)/XSIZEOF(Conveyor.aInverters[0])) - 1;
xInverterIndexOK := METH_IsValidInverterIndex(iIndex := TO_INT(uiInverterIndex));
xRangeValid := 
	METH_IsValidLocationIndex(iIndex := TO_INT(uiFrom))
	AND METH_IsValidLocationIndex(iIndex := TO_INT(uiTo))
	AND uiFrom <= uiTo
;
xParsingOK := 
	xInverterIndexOK
	AND xRangeValid
;

IF xParsingOK THEN
	FOR iInd := TO_INT(uiFrom) TO TO_INT(uiTo) DO
		Conveyor.aLocations[iInd].iInverterIndex := TO_INT(uiInverterIndex);
	END_FOR
ELSE
	iRes := -1;
END_IF

METH_SetInverterLocationsRange := iRes;

{warning enable C0371}

                
END_METHOD

(* For state monitoring and backup *)
METHOD METH_GetInternalState : BOOL
  VAR_OUTPUT
    aItems : ARRAY[0..GVL_Consts.gc_iMaxIndItems] OF items_struct_t;
  END_VAR
                  aItems := _aItemsStates;
                
END_METHOD

(* For state reconstruction after crash *)
METHOD METH_SetInternalState : BOOL
  VAR_OUTPUT
    aItems : ARRAY[0..GVL_Consts.gc_iMaxIndItems] OF items_struct_t;
  END_VAR
                  _aItemsStates := aItems;
                
END_METHOD
END_FUNCTION_BLOCK

FUNCTION_BLOCK FB_StanHome_Sorter01 EXTENDS FB_Sorter_TPL

            SUPER^(aBuffers := aBuffers, Conveyor := Conveyor);
uiErrorID := TO_UINT(_Model.iErrorID);
          

(* Must be called at least once. This method maps the interchange locations to move items between the conveyor and one of the buffers *)
METHOD METH_Map : INT
  VAR
    iInvLocRes : INT;
  END_VAR
                  {warning disable C0371}
ACT_HandleExternalContextWarning();

Conveyor.aLocations[1].iBufferIndex := 0; // shall be hard-coded depending on the physical implementation
Conveyor.aLocations[2].iBufferIndex := 1; // shall be hard-coded depending on the physical implementation
Conveyor.aLocations[3].iBufferIndex := 2;
Conveyor.aLocations[4].iBufferIndex := 3;

iInvLocRes := METH_SetInverterLocationsRange(
	uiInverterIndex := 0,
	uiFrom := 0,
	uiTo := 4
);

(**)
Conveyor.aLocations[5].iBufferIndex := 4; // shall be hard-coded depending on the physical implementation
Conveyor.aLocations[6].iBufferIndex := 5; // shall be hard-coded depending on the physical implementation
Conveyor.aLocations[7].iBufferIndex := 6;
Conveyor.aLocations[8].iBufferIndex := 7;

iInvLocRes := METH_SetInverterLocationsRange(
	uiInverterIndex := 1,
	uiFrom := 5,
	uiTo := 8
);


{warning enable C0371}

                
END_METHOD
END_FUNCTION_BLOCK

FUNCTION_BLOCK SQL_Interp_GetCommands EXTENDS SysD_DB.SQL_QueryInterpr_TPL

            
          

(* {warning 'Add method implementation '} *)
METHOD METH_GetNewKey : BOOL
  VAR_INPUT
    iInd : INT;
  END_VAR
  VAR_OUTPUT
    xwSize : __XWORD;
  END_VAR
  VAR
    pDestStruct : POINTER TO db_t_commands_struct_t;
    xRes : BOOL;
  END_VAR
                  pDestStruct := pSpecDestStruct;
CASE iInd OF
	0:
		sKey := 'id';
		pStartColumn := ADR(pDestStruct^.diID);
		VAR_INFO_ThisCol := __VARINFO(pDestStruct^.diID);
	1:
		sKey := 'source_position';
		pStartColumn := ADR(pDestStruct^.sSourcePosition);
		VAR_INFO_ThisCol := __VARINFO(pDestStruct^.sSourcePosition);
	2:
		sKey := 'destination_position';
		pStartColumn := ADR(pDestStruct^.sDestinationPosition);
		VAR_INFO_ThisCol := __VARINFO(pDestStruct^.sDestinationPosition);
	3:
		sKey := 'command_status';
		pStartColumn := ADR(pDestStruct^.iCommandStatus);
		VAR_INFO_ThisCol := __VARINFO(pDestStruct^.iCommandStatus);
	4:
		sKey := 'dt_inserted';
		pStartColumn := ADR(pDestStruct^.sInserted);
		VAR_INFO_ThisCol := __VARINFO(pDestStruct^.sInserted);
	5:
		sKey := 'dt_updated';
		pStartColumn := ADR(pDestStruct^.sUpdated);
		VAR_INFO_ThisCol := __VARINFO(pDestStruct^.sUpdated);
	6:
		xRes := TRUE;
END_CASE

xwSize := XSIZEOF(pDestStruct^); // must


METH_GetNewKey := xRes;
                
END_METHOD
END_FUNCTION_BLOCK

PROGRAM prgROS
  VAR_INPUT
    run_01 : BOOL;  (* to ROS *)
    run_02 : BOOL;
    lft_palletizing_options_01 : PalletizingOptions;
    lft_palletizing_options_02 : PalletizingOptions;
    rgt_palletizing_options_01 : PalletizingOptions;
    rgt_palletizing_options_02 : PalletizingOptions;
    lifter_controller_feedback_01 : CommonFeedback;
    lifter_controller_feedback_02 : CommonFeedback;
    lifter_controller_joint_states_01 : JointState;
    lifter_controller_joint_states_02 : JointState;
  END_VAR
  VAR_OUTPUT
    process_code_01 : DINT;  (* to codesys *)
    process_code_02 : DINT;
    lifter_controller_command_01 : CommonCommand;
    lifter_controller_command_02 : CommonCommand;
  END_VAR
  VAR
    ROSInterface_01 : ros_interface_struct_t;
    ROSInterface_02 : ros_interface_struct_t;
    robin : Robin;
    sState : STRING(255) := 'Boolean tests';
    xTB_Mode : BOOL;
    xENInv_Mode : BOOL;
    xEnableCount : BOOL := TRUE;
    xSafetyCondOK : BOOL := TRUE;
    xEN_ROSCommands : BOOL;
    xENInv_ROSCommands : BOOL;
    R_TRIG_Run : R_TRIG;
    xProposedFlip : BOOL;
    iTotalHistory : INT;
    iMinHistoryNum : INT := 5;
    aTON_VisionNotArriving : ARRAY[0..1] OF TON;
    atLoaded : ARRAY[0..1] OF TIME := [2(TIME#40s0ms)];
    axVisionNotArrivingCond : ARRAY[0..1] OF BOOL;
    xPieceErrorCond : BOOL;
    xResetErrorCond : BOOL;
    xBypassReset : BOOL := TRUE;
    xResetFlipAtMachineReset : BOOL;
    xROSIsResetCond : BOOL;
    R_TRIG_Resetting : R_TRIG;
    xAutoFlipping : BOOL := TRUE;
    lrPercNOT_OK : LREAL;
    xTB_CleanHistory : BOOL;
    diProcessCode : DINT;
    xEN_ROSRun : BOOL;  (* xSafetyCondOK: BOOL; *)
    xENInv_ROSRun : BOOL;
    eROSMode : device_mode_enum_t;
    xEnableCountInManualMode : BOOL;
    dwFontColorID : DWORD;  (* xEN_ROSCommands: BOOL; *)
    R_TRIG_ROSErrorDetected_01 : R_TRIG;  (* xThereIsROSError : BOOL; *)
    R_TRIG_ROSErrorDetected_02 : R_TRIG;
    xROSErrorMonitoring : BOOL;
    xSafetyAlwaysON : BOOL;
    R_TRIG_PickError : R_TRIG;
    iPickAttempts : INT;
    iPlaceAttempts : INT;
    diProcessCode_01 : DINT;
    xThereIsROSError_01 : BOOL;
    diProcessCode_02 : DINT;
    xThereIsROSError_02 : BOOL;
    eProcessState_01 : process_code_enum_t;
    lwSubSize : LWORD;
    lwPubSize : LWORD;
    udiResProcEnter : RTS_IEC_RESULT;
    udiResProcLeave : RTS_IEC_RESULT;
    sPatternFolderPath : STRING(255);
  END_VAR

                    // instancing Robin class
robin();

//////////////////////////////////////////////////////////////////////////////////////////////////////////////////////////////////////////
//																																		//
//												READ - robin.read(<topic_name>, <variable>)												//
//																																		//
//////////////////////////////////////////////////////////////////////////////////////////////////////////////////////////////////////////

robin.read('process_code_01', process_code_01);
robin.read('process_code_02', process_code_02);

robin.read('lifter_controller_command_01', lifter_controller_command_01);
robin.read('lifter_controller_command_02', lifter_controller_command_02);

//////////////////////////////////////////////////////////////////////////////////////////////////////////////////////////////////////////
//																																		//
//												WRITE - robin.write(<topic_name>, <variable>)											//
//																																		//
//////////////////////////////////////////////////////////////////////////////////////////////////////////////////////////////////////////

robin.write('run_01', run_01);
robin.write('run_02', run_02);

robin.write('lft_palletizing_options_01', lft_palletizing_options_01);
robin.write('lft_palletizing_options_02', lft_palletizing_options_02);

robin.write('rgt_palletizing_options_01', rgt_palletizing_options_01);
robin.write('rgt_palletizing_options_02', rgt_palletizing_options_02);

robin.write('lifter_controller_feedback_01', lifter_controller_feedback_01);
robin.write('lifter_controller_feedback_02', lifter_controller_feedback_02);

robin.write('lifter_controller_joint_states_01', lifter_controller_joint_states_01);
robin.write('lifter_controller_joint_states_02', lifter_controller_joint_states_02);

//////////////////////////////////////////////////////////////////////////////////////////////////////////////////////////////////////////
// SHARED MEMORY VARIABLES

// IMPORT VALUES FROM SUBSCRIPTIONS
ACT_ImportSubValues_01();
ACT_ImportSubValues_02();

(*----------------------------------------------------------------*)
(* EXPORT VALUES TO PUBLICATIONS *)
ACT_ExportPubValues_01();
ACT_ExportPubValues_02();

(*----------------------------------------------------------------*)
(*----------------------------------------------------------------*)
(*----------------------------------------------------------------*)
// FURTHER EVALUATIONS

// RICOSTRUZIONE PROCESS STATE
ACT_ProcessState01();
ACT_ProcessState02();


ACT_ErrorMonitoring01();
// ACT_ErrorMonitoring01();
(*-----------------------------------------------------------------*)
ACT_Mode();




                  

ACTION ACT_ResetVision:
                        GVL.g_ROSInterface.aObjectManager[iInd].xResult_OK := FALSE;
		GVL.g_ROSInterface.aObjectManager[iInd].xResult_NOT_OK := FALSE;
		GVL_Applica.g_MachineMESInterface.Details.aPieces[iInd].eState := piece_state_enum_t.PieceUnknownState;
                      
END_ACTION

ACTION ACT_ProcessState01:
                        diProcessCode_01 := ROSInterface_01.ROS2Codesys.Subscripted.process_code;
ROSInterface_01.ROS2Codesys.eProcessState := METH_GetProcessState(
	diProcessCode := diProcessCode_01
);
(*----------------------------*)
// BT error detection
xThereIsROSError_01 := diProcessCode_01 < 0;
R_TRIG_ROSErrorDetected_01(CLK := xThereIsROSError_01);
IF R_TRIG_ROSErrorDetected_01.Q THEN
	METH_SetRun_01(xValue := FALSE);
	xROSErrorMonitoring := TRUE;
	xSafetyAlwaysON := GVL.g_xSafetyOK;
END_IF
                      
END_ACTION

ACTION ACT_ProcessState02:
                        diProcessCode_02 := ROSInterface_02.ROS2Codesys.Subscripted.process_code;
ROSInterface_02.ROS2Codesys.eProcessState := METH_GetProcessState(
	diProcessCode := diProcessCode_02
);
(*----------------------------*)
// BT error detection
xThereIsROSError_02 := diProcessCode_02 < 0;
R_TRIG_ROSErrorDetected_02(CLK := xThereIsROSError_02);
IF R_TRIG_ROSErrorDetected_02.Q THEN
	METH_SetRun_02(xValue := FALSE);
	xROSErrorMonitoring := TRUE;
	xSafetyAlwaysON := GVL.g_xSafetyOK;
END_IF
                      
END_ACTION

ACTION ACT_ErrorMonitoring01:
                        (*----------------------------*)
IF NOT (xThereIsROSError_01 OR xThereIsROSError_02) THEN
	xROSErrorMonitoring := FALSE;
END_IF
(*----------------------------*)
// BT pick error counter
eProcessState_01 := ROSInterface_01.ROS2Codesys.eProcessState;
R_TRIG_PickError(CLK := eProcessState_01 = process_code_enum_t.pcode_PickError);
IF R_TRIG_PickError.Q THEN
	METH_IncrementPickErrorCounter();
END_IF

                      
END_ACTION

ACTION ACT_Mode:
                        xENInv_Mode := FALSE;
IF xTB_Mode THEN
	eROSMode := device_mode_enum_t.MANUAL_MODE;
ELSE
	eROSMode := device_mode_enum_t.AUTOMATIC_MODE;
END_IF
(*-----------------------------------------------------------------*)
xEN_ROSRun := xSafetyCondOK;
xENInv_ROSRun := NOT xEN_ROSRun;

// xEN_ROSCommands := run_01;
xENInv_ROSCommands := NOT xEN_ROSCommands;

(*-----------------------------------------------------------------*)
// MODE
CASE eROSMode OF
	device_mode_enum_t.AUTOMATIC_MODE:
		//
		xEnableCount := TRUE;
	(*------------------------------------------------------------*)
	device_mode_enum_t.MANUAL_MODE:
		//
		xEnableCount := xEnableCountInManualMode;
	(*------------------------------------------------------------*)
END_CASE
(*-----------------------------------------------------------------*)
// COMMANDS
R_TRIG_Run(CLK := GVL.g_xRUNNING);
IF R_TRIG_Run.Q THEN // partenza
	//
	eROSMode := device_mode_enum_t.AUTOMATIC_MODE;
END_IF

                      
END_ACTION

ACTION ACT_ExportPubValues_01:
                        run_01 := ROSInterface_01.Codesys2ROS.Published.run;
lft_palletizing_options_01 := ROSInterface_01.Codesys2ROS.Published.lft_palletizing_options;
rgt_palletizing_options_01 := ROSInterface_01.Codesys2ROS.Published.rgt_palletizing_options;
lifter_controller_feedback_01 := ROSInterface_01.Codesys2ROS.Published.lifter_controller_feedback;
lifter_controller_joint_states_01 := ROSInterface_01.Codesys2ROS.Published.lifter_controller_joint_states;
                      
END_ACTION

ACTION ACT_ImportSubValues_01:
                        ROSInterface_01.ROS2Codesys.Subscripted.process_code := process_code_01;
ROSInterface_01.ROS2Codesys.Subscripted.lifter_controller_command := lifter_controller_command_01;
                      
END_ACTION

ACTION ACT_ExportPubValues_02:
                        run_02 := ROSInterface_02.Codesys2ROS.Published.run;
lft_palletizing_options_02 := ROSInterface_02.Codesys2ROS.Published.lft_palletizing_options;
rgt_palletizing_options_02 := ROSInterface_02.Codesys2ROS.Published.rgt_palletizing_options;
lifter_controller_feedback_02 := ROSInterface_02.Codesys2ROS.Published.lifter_controller_feedback;
lifter_controller_joint_states_02 := ROSInterface_02.Codesys2ROS.Published.lifter_controller_joint_states;
                      
END_ACTION

ACTION ACT_ImportSubValues_02:
                        ROSInterface_02.ROS2Codesys.Subscripted.process_code := process_code_02;
ROSInterface_02.ROS2Codesys.Subscripted.lifter_controller_command := lifter_controller_command_02;
                      
END_ACTION

METHOD METH_IncrementPickErrorCounter : BOOL
                          iPickAttempts := iPickAttempts + 1;
                        
END_METHOD

METHOD METH_ResetPickErrorCounter : BOOL
                          iPickAttempts := 0;
                        
END_METHOD

METHOD METH_IncrementPlaceErrorCounter : BOOL
                          iPickAttempts := iPickAttempts + 1;
                        
END_METHOD

METHOD METH_ResetPlaceErrorCounter : BOOL
                          iPlaceAttempts := 0;
                        
END_METHOD

METHOD METH_GetProcessState : process_code_enum_t
  VAR_INPUT
    diProcessCode : DINT;
  END_VAR
  VAR
    eRes : process_code_enum_t;
  END_VAR
                          IF diProcessCode >= 0 THEN // Process OK	
	IF diProcessCode = 0 THEN
		eRes := process_code_enum_t.pcode_ToInitialize;	
	ELSIF diProcessCode = GVL_ProcessCode.gc_diPICK_RUNNING THEN
		eRes := process_code_enum_t.pcode_PickRunning;	
	ELSIF diProcessCode = GVL_ProcessCode.gc_diPLACE_RUNNING THEN
		eRes := process_code_enum_t.pcode_PlaceRunning;	
	ELSIF diProcessCode = GVL_ProcessCode.gc_diFINISHED THEN
		eRes := process_code_enum_t.pcode_Finished;	
	ELSE
		eRes := process_code_enum_t.pcode_Unknown;
	END_IF
ELSE // errors
	CASE diProcessCode OF
		GVL_ProcessCode.gc_diPICK_FAILED:
			eRes := process_code_enum_t.pcode_PickError;
		GVL_ProcessCode.gc_diPLACE_FAILED:
			eRes := process_code_enum_t.pcode_PlaceError;
		ELSE
			eRes := process_code_enum_t.pcode_Error;
	END_CASE
END_IF

METH_GetProcessState := eRes;
                        
END_METHOD

METHOD METH_SetRun_01 : BOOL
  VAR_INPUT
    xValue : BOOL;
  END_VAR
                          ROSInterface_01.Codesys2ROS.Published.run := xValue;

METH_SetRun_01 := ROSInterface_01.Codesys2ROS.Published.run;
                        
END_METHOD

METHOD METH_SetRun_02 : BOOL
  VAR_INPUT
    xValue : BOOL;
  END_VAR
                          ROSInterface_02.Codesys2ROS.Published.run := xValue;

METH_SetRun_02 := ROSInterface_02.Codesys2ROS.Published.run;
                        
END_METHOD

METHOD METH_SetObjectName_Left_01
  VAR_INPUT
    sValue : STRING;
  END_VAR
                          ROSInterface_01.Codesys2ROS.Published.lft_palletizing_options.object_name := sValue;
                        
END_METHOD

METHOD METH_SetObjectName_Right_01
  VAR_INPUT
    sValue : STRING;
  END_VAR
                          ROSInterface_01.Codesys2ROS.Published.rgt_palletizing_options.object_name := sValue;
                        
END_METHOD

METHOD METH_SetObjectName_Left_02
  VAR_INPUT
    sValue : STRING;
  END_VAR
                          ROSInterface_02.Codesys2ROS.Published.lft_palletizing_options.object_name := sValue;
                        
END_METHOD

METHOD METH_SetObjectName_Right_02
  VAR_INPUT
    sValue : STRING;
  END_VAR
                          ROSInterface_02.Codesys2ROS.Published.rgt_palletizing_options.object_name := sValue;
                        
END_METHOD

METHOD METH_SetObjectWeight_Left_01
  VAR_INPUT
    lrValue : LREAL;
  END_VAR
                          ROSInterface_01.Codesys2ROS.Published.lft_palletizing_options.object_weight := lrValue;
                        
END_METHOD

METHOD METH_SetObjectWeight_Right_01
  VAR_INPUT
    lrValue : LREAL;
  END_VAR
                          ROSInterface_01.Codesys2ROS.Published.rgt_palletizing_options.object_weight := lrValue;
                        
END_METHOD

METHOD METH_SetObjectWeight_Left_02
  VAR_INPUT
    lrValue : LREAL;
  END_VAR
                          ROSInterface_02.Codesys2ROS.Published.lft_palletizing_options.object_weight := lrValue;
                        
END_METHOD

METHOD METH_SetObjectWeight_Right_02
  VAR_INPUT
    lrValue : LREAL;
  END_VAR
                          ROSInterface_02.Codesys2ROS.Published.rgt_palletizing_options.object_weight := lrValue;
                        
END_METHOD

METHOD METH_SetPatternName_Left_01
  VAR_INPUT
    sValue : STRING;
  END_VAR
                          ROSInterface_01.Codesys2ROS.Published.lft_palletizing_options.pattern_file := METH_ComposePatternFilePath(
	sPatternName := sValue
);
                        
END_METHOD

METHOD METH_SetPatternName_Right_01
  VAR_INPUT
    sValue : STRING;
  END_VAR
                          ROSInterface_01.Codesys2ROS.Published.rgt_palletizing_options.pattern_file := METH_ComposePatternFilePath(
	sPatternName := sValue
);
                        
END_METHOD

METHOD METH_SetTransform_Right_01
  VAR_INPUT
    sValue : STRING;
  END_VAR
                          ROSInterface_01.Codesys2ROS.Published.rgt_palletizing_options.transform_name := sValue;
                        
END_METHOD

METHOD METH_SetTransform_Left_02
  VAR_INPUT
    sValue : STRING;
  END_VAR
                          ROSInterface_02.Codesys2ROS.Published.lft_palletizing_options.transform_name := sValue;
                        
END_METHOD

METHOD METH_SetPatternName_Left_02
  VAR_INPUT
    sValue : STRING;
  END_VAR
                          ROSInterface_02.Codesys2ROS.Published.lft_palletizing_options.pattern_file := METH_ComposePatternFilePath(
	sPatternName := sValue
);
                        
END_METHOD

METHOD METH_SetPatternName_Right_02
  VAR_INPUT
    sValue : STRING;
  END_VAR
                          ROSInterface_02.Codesys2ROS.Published.rgt_palletizing_options.pattern_file := METH_ComposePatternFilePath(
	sPatternName := sValue
);
                        
END_METHOD

METHOD METH_ComposePatternFilePath : STRING(255)
  VAR_INPUT
    sPatternName : STRING;
  END_VAR
  VAR
    sRes : STRING(255);
  END_VAR
                          sRes :=
	CONCAT(
		sPatternFolderPath,
		CONCAT(
			sPatternName,
			'.yaml'
		)
	)
;

METH_ComposePatternFilePath := sRes;
                        
END_METHOD

METHOD METH_SetTransform_Left_01
  VAR_INPUT
    sValue : STRING;
  END_VAR
                          ROSInterface_01.Codesys2ROS.Published.lft_palletizing_options.transform_name := sValue;
                        
END_METHOD

METHOD METH_SetTransform_Right_02
  VAR_INPUT
    sValue : STRING;
  END_VAR
                          ROSInterface_02.Codesys2ROS.Published.rgt_palletizing_options.transform_name := sValue;
                        
END_METHOD

METHOD METH_SetToolName_Left_01
  VAR_INPUT
    sValue : STRING;
  END_VAR
                          ROSInterface_01.Codesys2ROS.Published.lft_palletizing_options.tool_name := sValue;
                        
END_METHOD

METHOD METH_SetToolName_Right_01
  VAR_INPUT
    sValue : STRING;
  END_VAR
                          ROSInterface_01.Codesys2ROS.Published.rgt_palletizing_options.tool_name := sValue;
                        
END_METHOD

METHOD METH_SetToolName_Left_02
  VAR_INPUT
    sValue : STRING;
  END_VAR
                          ROSInterface_02.Codesys2ROS.Published.lft_palletizing_options.tool_name := sValue;
                        
END_METHOD

METHOD METH_SetToolName_Right_02
  VAR_INPUT
    sValue : STRING;
  END_VAR
                          ROSInterface_02.Codesys2ROS.Published.rgt_palletizing_options.tool_name := sValue;
                        
END_METHOD
END_PROGRAM

PROGRAM prgMain
  VAR
    sHostName : STRING;
    eProposedMachineState : machine_state_enum_t;
    eProposedMachineError : machine_error_enum_t;
    eStep : step_enum_t;  (* xPausedWhileRunning: BOOL; *)
    iStepInit : INT;
    xInitialize : BOOL;
    xInitialized : BOOL;
    xInitError : BOOL;
    TON_WaitBTOn : TON;
    tWaitBT : TIME := TIME#5s0ms;
    F_TRIG_Pause : F_TRIG;
    xErrorStopAck : BOOL := TRUE;
    TON_ListDockers : TON;
    tListDockersPolling : TIME := TIME#5s0ms;
    xStartBTCOnd : BOOL;
    xStartDoosanCond : BOOL;
    xBTIsActive : BOOL;
    xDisableRUN_DebugFlag : BOOL := FALSE;
    xRestartAllCond : BOOL;
    xJustRestartBTCond : BOOL;
    xJustBTOff : BOOL;
    xEverythingOoffCond : BOOL;
    xDoosanOkButBTOff : BOOL;
    xARunWasGiven : BOOL;
    xPalletTerminated : BOOL;
    R_TRIG_JustTerminated : R_TRIG;
    xDormantCond : BOOL;
    xStartCond : BOOL;
    xVisionCond : BOOL;
    xPickCond : BOOL;
    xPlaceCond : BOOL;
    xPickErrorCond : BOOL;
    xPlaceErrorCond : BOOL;
    xCycleFinished : BOOL;
    xToInit : BOOL;
    eProcessState_01 : process_code_enum_t;
  END_VAR

                    // MAIN COMMANDS
IF GVL.g_xPLAY THEN
	GVL.g_xPLAY := FALSE;
	GVL.g_xRUNNING := TRUE;
	xInitialize := TRUE;
	xARunWasGiven := FALSE;
END_IF

ACT_Initialize();

IF GVL.g_xPAUSE AND GVL.g_xRUNNING THEN //06/06/2022
	prgROS.METH_SetRun_01(xValue := FALSE);
// 	GVL.g_ROSInterface_01.xRun := FALSE;
// 	xPausedWhileRunning := TRUE;
END_IF

IF GVL.g_xRUNNING THEN
	F_TRIG_Pause(CLK := GVL.g_xPAUSE);
	IF F_TRIG_Pause.Q THEN
		prgROS.METH_SetRun_01(xValue := TRUE);
// 		GVL.g_ROSInterface_01.xRun := TRUE;
	END_IF
END_IF



IF GVL.g_xRESET THEN
	GVL.g_xRESET := FALSE;
	GVL_HMI.g_xIsStoppedByUser := FALSE;
	
// 	GVL.g_xNODES_START := TRUE;
	GVL.g_xRESETTING := TRUE;
	
	GVL.g_xRUNNING := FALSE;
// 	GVL.g_xPAUSE := FALSE;
	GVL_HMI.xPause := FALSE;
END_IF

IF GVL.g_xSTOP THEN
	GVL.g_xSTOP := FALSE;
	GVL.g_xRUNNING := FALSE;
// 	GVL.g_xPAUSE := FALSE;
	GVL_HMI.xPause := FALSE;
// 	GVL.g_xNODES_STOP := TRUE;
	IF NOT prgLinuxCommand.METH_IsDockerBTActive_01() AND NOT prgLinuxCommand.METH_IsDockerBTActive_02() THEN
		prgLinuxCommand.METH_StopAllDockers();
	ELSE
		IF prgLinuxCommand.METH_IsDockerBTActive_01() THEN
			prgLinuxCommand.METH_StopBT01();
		END_IF
		IF prgLinuxCommand.METH_IsDockerBTActive_02() THEN
			prgLinuxCommand.METH_StopBT02();
		END_IF
	END_IF
	xInitialized := FALSE;
	xErrorStopAck := FALSE;
	xARunWasGiven := FALSE;
END_IF

IF GVL.g_xRESETTING THEN
	eStep := step_enum_t.Dormant;
	GVL.g_xRESETTING := FALSE;
	xErrorStopAck := TRUE;
END_IF
(*-----------------------------------------------------------------*)

(*-----------------------------------------------------------------*)
// MACHINE STATE
METH_GetMachineState(eState => eProposedMachineState, eError => eProposedMachineError);
GVL_Applica.g_MachineMESInterface.Machine.eState := eProposedMachineState;
GVL_Applica.g_MachineMESInterface.Machine.eError := eProposedMachineError;
(*-----------------------------------------------------------------*)

SysSocket.SysSockGetHostName(diNameLen := TO_DINT(XSIZEOF(sHostName)), szHostName := sHostName);
GVL.g_xLocalTestMachine := sHostName = 'gazelle';

GVL_HMI.xTowerLight_Red := GVL.g_LightTower.xRed;
GVL_HMI.xTowerLight_Yellow := GVL.g_LightTower.xYellow;
GVL_HMI.xTowerLight_Green := GVL.g_LightTower.xGreen;
(*-----------------------------------------------------------------*)

xPalletTerminated := eStep = step_enum_t.Terminated;
R_TRIG_JustTerminated(CLK := xPalletTerminated);
IF R_TRIG_JustTerminated.Q THEN
	prgROS.METH_SetRun_01(xValue := FALSE);
// 	GVL.g_ROSInterface_01.xRun := FALSE;
END_IF

// seguo ciclo BT
eProcessState_01 := prgROs.ROSInterface_01.ROS2Codesys.eProcessState;
xDormantCond := METH_DetectDormant(eProcStat := eProcessState_01);
xStartCond := METH_DetectStart(eProcStat := eProcessState_01);
xVisionCond := METH_DetectVision(eProcStat := eProcessState_01);
xPickCond := METH_DetectPick(eProcStat := eProcessState_01);
xPlaceCond := METH_DetectPlace(eProcStat := eProcessState_01);
xPickErrorCond := METH_DetectPickError(eProcStat := eProcessState_01);
xPlaceErrorCond := METH_DetectPlaceError(eProcStat := eProcessState_01);
xCycleFinished := METH_DetectFinished(eProcStat := eProcessState_01);

// CYCLE
CASE eStep OF
	step_enum_t.Dormant:
		xToInit := NOT xInitialized;
		IF xStartCond THEN
			IF xVisionCond THEN
				eStep := step_enum_t.Vision;
			ELSIF xPickCond THEN
				eStep := step_enum_t.Pick;
			ELSIF xPlaceCond THEN
				eStep := step_enum_t.Place;
			END_IF
		END_IF
	(*-------------------------------------*)
	step_enum_t.Vision: //03/05/2023
		IF xPickCond THEN
			eStep := step_enum_t.Pick;
		END_IF
	(*-------------------------------------*)
	step_enum_t.Pick:
		IF xPickErrorCond THEN
			eStep := step_enum_t.Error;
		ELSIF xPlaceCond THEN
			eStep := step_enum_t.Place;
		END_IF
	(*-------------------------------------*)
	step_enum_t.Place:
		IF xPlaceErrorCond THEN
			eStep := step_enum_t.Error;
		ELSIF xCycleFinished THEN
			eStep := step_enum_t.Terminated;
		ELSIF xPickCond THEN
			eStep := step_enum_t.Pick;
		ELSIF xDormantCond THEN
			eStep := step_enum_t.Dormant;
		END_IF
	(*-------------------------------------*)
	step_enum_t.Terminated:
// 		IF METH_DetectDormant() THEN
		eStep := step_enum_t.Dormant;
		prgROS.METH_ResetPickErrorCounter();
		prgROS.METH_ResetPlaceErrorCounter();
// 		END_IF
	(*-------------------------------------*)
	step_enum_t.Error:
		IF xStartCond THEN
			IF xPickCond THEN
				eStep := step_enum_t.Vision;
			ELSIF xPickCond THEN
				eStep := step_enum_t.Pick;
			ELSIF xPlaceCond THEN
				eStep := step_enum_t.Place;
			END_IF
		ELSIF xDormantCond AND xInitialized THEN
			eStep := step_enum_t.Dormant;
			prgROS.METH_ResetPickErrorCounter();
			prgROS.METH_ResetPlaceErrorCounter();
		END_IF
	(*-------------------------------------*)
END_CASE
(*----------------------------------*)
TON_ListDockers(IN := NOT prgLinuxCommand.xDIS_Command, PT := tListDockersPolling);
IF TON_ListDockers.Q THEN
	TON_ListDockers(IN := FALSE);
	prgLinuxCommand.METH_ListDockers();
END_IF
                  

ACTION ACT_Initialize:
                        CASE iStepInit OF
	0:
		TON_WaitBTOn(IN := FALSE);
		IF xInitialize THEN
			xInitialize := FALSE;
			IF METH_IsGazelle() THEN
				iStepInit := 4;
			ELSE
				xJustRestartBTCond := METH_IsJustRestartBT();
				xRestartAllCond := METH_IsRestartAll();
				xEverythingOoffCond := METH_IsEveryThingOff();
				xDoosanOkButBTOff := METH_IsDoosanOkButBTOff();
				IF xDoosanOkButBTOff THEN
					iStepInit := 2;
				ELSIF xRestartAllCond THEN
					iStepInit := 1;
					prgLinuxCommand.METH_StopAllDockers(); // stop all
				ELSIF xJustRestartBTCond THEN
					iStepInit := 11;
					IF prgLinuxCommand.METH_IsDockerBTActive_01() THEN
						prgLinuxCommand.METH_StopBT01();
					END_IF
					IF prgLinuxCommand.METH_IsDockerBTActive_02() THEN
						prgLinuxCommand.METH_StopBT02();
					END_IF
				ELSIF xEverythingOoffCond THEN // alerady everything off
					prgLinuxCommand.METH_StartDoosanDocker();
					iStepInit := 2;
				ELSE
					xInitError := TRUE;
				END_IF
			END_IF
		END_IF		
	(*----------------------------*)
	1: // start doosan
		xStartDoosanCond := 
			prgEIPMapping.METH_IsDoosanSafeOff(DoosanState := prgEIPMapping.DoosanState)
			AND NOT prgLinuxCommand.METH_IsDockerDoosanActive()
			AND NOT prgLinuxCommand.METH_IsDockerBTActive()
		;
		IF xStartDoosanCond THEN
			prgLinuxCommand.METH_StartDoosanDocker(); // start doosan
			iStepInit := 2;
		END_IF
	(*----------------------------*)
	11: // just bt off
		xJustBTOff := 
			NOT prgLinuxCommand.METH_IsDockerBTActive()
		;
		IF xJustBTOff THEN
			iStepInit := 2;
		END_IF
	(*----------------------------*)
	2: // start bt
		xStartBTCOnd := 
			prgEIPMapping.METH_IsDoosanServoOn(DoosanState := prgEIPMapping.DoosanState)
		;
		IF xStartBTCOnd THEN
			xInitError := FALSE;
			IF METH_IsPalletConfig01() THEN
				prgLinuxCommand.METH_StartBT01();
			ELSIF METH_IsPalletConfig02() THEN
				prgLinuxCommand.METH_StartBT02();
			ELSE
				xInitError := TRUE;
			END_IF
			IF NOT xInitError THEN
				iStepInit := iStepInit + 1;
			END_IF
		END_IF
	(*----------------------------*)
	3: // wait finished
		TON_WaitBTOn(IN := TRUE, PT := tWaitBT);
		xBTIsActive := prgLinuxCommand.METH_IsDockerBTActive();
		IF (TON_WaitBTOn.Q AND xBTIsActive) OR xBTIsActive THEN
			TON_WaitBTOn(IN := FALSE);
			iStepInit := iStepInit + 1;
		END_IF
	(*----------------------------*)
	4: // end
		xInitialized := TRUE;
		iStepInit := 0;
		IF NOT xDisableRUN_DebugFlag THEN
			prgROS.METH_SetRun_01(xValue := TRUE);
// 			GVL.g_ROSInterface_01.xRun := TRUE;
			xARunWasGiven := TRUE;
		END_IF
	(*----------------------------*)
END_CASE
                      
END_ACTION

METHOD METH_GetMachineState
  VAR_INPUT
    iIndex : INT := 1;
  END_VAR
  VAR_OUTPUT
    eState : machine_state_enum_t := machine_state_enum_t.MachineUnknownState;
    eError : machine_error_enum_t := machine_error_enum_t.NO_ERROR;
  END_VAR
  VAR
    xSafetyCondOK : BOOL;
    xPaused : BOOL;
    xInError : BOOL;
    xRun : BOOL;
    iMaxInd : INT;
    iInd : INT := 0;
    xObjInError : BOOL;
    xAMRInError : BOOL;
    xToInit : BOOL;
    xResetting : BOOL;
    xVisionError : BOOL;
    xVisionWarning : BOOL;
    xBTError : BOOL;
    xInitializing : BOOL;
    xInvalidInputError : BOOL;
  END_VAR
                          
CASE iIndex OF
	1:
		xBTError := prgROS.ROSInterface_01.ROS2Codesys.Subscripted.process_code < 0 AND NOT xErrorStopAck;
	2:
		xBTError := prgROS.ROSInterface_01.ROS2Codesys.Subscripted.process_code < 0 AND NOT xErrorStopAck;
	ELSE
		xInvalidInputError := TRUE;
		xBTError := FALSE;
END_CASE


xInError := 
	xObjInError 
	OR GVL.g_xRobotError 
	OR GVL.g_xPieceError 
	OR GVL_HMI.g_xIsStoppedByUser 
	OR xBTError
	OR xInvalidInputError
;

xResetting := GVL.g_xRESETTING;
xInitializing := METH_DetectInitializing();
xToInit := xInitializing;





// xToInit := GVL_EasySolution.g_MachineMESInterface.Details.Fleet.eState = fleet_state_enum_t.TO_INITIALIZE;

xRun := GVL.g_xRUNNING;
xSafetyCondOK := GVL.g_xSafetyOK AND GVL.g_xSafeguardOK;

IF xInvalidInputError THEN
	eState := machine_state_enum_t.MachineUnknownState;
	eError := machine_error_enum_t.GENERAL_ERROR;
ELSIF NOT xSafetyCondOK THEN
	IF GVL.g_xSafetyOK THEN
		eState := machine_state_enum_t.MachineSafeguardStop;
	ELSE
		eState := machine_state_enum_t.MachineSafetyStop;
	END_IF
	eError := machine_error_enum_t.EM_STOP;
ELSE
	IF xResetting THEN
		eState := machine_state_enum_t.MachineReset;
	ELSIF xVisionError THEN
		eState := machine_state_enum_t.MachineError;
		eError := machine_error_enum_t.CAMERA_ERROR;
	ELSIF xVisionWarning THEN
		eState := machine_state_enum_t.MachineWarning;
		eError := machine_error_enum_t.CAMERA_ERROR;
	ELSIF xInError THEN
		eState := machine_state_enum_t.MachineError;
		IF GVL.g_xPieceError THEN
			eError := machine_error_enum_t.PIECE_NOT_FOUND;
		ELSIF GVL_HMI.g_xIsStoppedByUser THEN //24/11/2022
			eError := machine_error_enum_t.STOPPED_BY_USER;
		ELSIF xBTError THEN
			eError := machine_error_enum_t.EXECUTION_ERROR;
		ELSE
			eError := machine_error_enum_t.GENERAL_ERROR;
		END_IF
	ELSIF xToInit THEN
		eState := machine_state_enum_t.MachineToInitialize;
	ELSE
		IF GVL.g_xPAUSE THEN
			eState := machine_state_enum_t.MachinePaused;
		ELSE
			IF xRun THEN
				eState := machine_state_enum_t.MachineRunning;
			ELSE
				eState := machine_state_enum_t.MachineReady;
			END_IF
		END_IF
		
	END_IF
END_IF
                        
END_METHOD

METHOD METH_DetectStart : BOOL
  VAR_INPUT
    eProcStat : process_code_enum_t;
  END_VAR
                          METH_DetectStart := 
	(
		METH_DetectVision(eProcStat := eProcStat) 
		OR METH_DetectPick(eProcStat := eProcStat) 
		OR METH_DetectPlace(eProcStat := eProcStat)
	) AND xInitialized
;
                        
END_METHOD

METHOD METH_DetectPick : BOOL
  VAR_INPUT
    eProcStat : process_code_enum_t;
  END_VAR
                          METH_DetectPick := eProcStat = process_code_enum_t.pcode_PickRunning;
                        
END_METHOD

METHOD METH_DetectPlace : BOOL
  VAR_INPUT
    eProcStat : process_code_enum_t;
  END_VAR
                          METH_DetectPlace := eProcStat = process_code_enum_t.pcode_PlaceRunning;
                        
END_METHOD

METHOD METH_DetectPickError : BOOL
  VAR_INPUT
    eProcStat : process_code_enum_t;
  END_VAR
                          METH_DetectPickError := eProcStat = process_code_enum_t.pcode_PickError;
                        
END_METHOD

METHOD METH_DetectPlaceError : BOOL
  VAR_INPUT
    eProcStat : process_code_enum_t;
  END_VAR
                          METH_DetectPlaceError := eProcStat = process_code_enum_t.pcode_PlaceError;
                        
END_METHOD

METHOD METH_DetectDormant : BOOL
  VAR_INPUT
    eProcStat : process_code_enum_t;
  END_VAR
                          METH_DetectDormant := eProcStat = process_code_enum_t.pcode_ToInitialize;
                        
END_METHOD

METHOD METH_DetectFinished : BOOL
  VAR_INPUT
    eProcStat : process_code_enum_t;
  END_VAR
                          METH_DetectFinished := eProcStat = process_code_enum_t.pcode_Finished;
                        
END_METHOD

METHOD METH_SetPalletConfig01
                          PersVars.g_uiCurrentPalletConfig := GVL_Constants.gc_uiPalletConfigIndex_01;
                        
END_METHOD

METHOD METH_SetPalletConfig02
                          PersVars.g_uiCurrentPalletConfig := GVL_Constants.gc_uiPalletConfigIndex_02;
                        
END_METHOD

METHOD METH_IsPalletConfig01 : BOOL
                          METH_IsPalletConfig01 := PersVars.g_uiCurrentPalletConfig = GVL_Constants.gc_uiPalletConfigIndex_01;
                        
END_METHOD

METHOD METH_IsPalletConfig02 : BOOL
                          METH_IsPalletConfig02 := PersVars.g_uiCurrentPalletConfig = GVL_Constants.gc_uiPalletConfigIndex_02;
                        
END_METHOD

METHOD METH_IsGazelle : BOOL
                          METH_IsGazelle := sHostName = 'gazelle';
                        
END_METHOD

METHOD METH_IsJustRestartBT : BOOL
                          METH_IsJustRestartBT := 
	prgLinuxCommand.METH_IsDockerBTActive()
	AND prgLinuxCommand.METH_IsDockerDoosanActive()
	AND prgEIPMapping.METH_IsDoosanServoOn(DoosanState := prgEIPMapping.DoosanState)
;
                        
END_METHOD

METHOD METH_IsRestartAll : BOOL
                          METH_IsRestartAll := 
	prgLinuxCommand.METH_IsDockerBTActive()
	AND prgLinuxCommand.METH_IsDockerDoosanActive()
	AND NOT prgEIPMapping.METH_IsDoosanServoOn(DoosanState := prgEIPMapping.DoosanState)
;
                        
END_METHOD

METHOD METH_IsEverythingOff : BOOL
                          METH_IsEverythingOff := 
	NOT prgLinuxCommand.METH_IsDockerBTActive()
	AND NOT prgLinuxCommand.METH_IsDockerDoosanActive()
	AND NOT prgEIPMapping.METH_IsDoosanServoOn(DoosanState := prgEIPMapping.DoosanState)
;
                        
END_METHOD

METHOD METH_IsDoosanOkButBTOff : BOOL
                          METH_IsDoosanOkButBTOff := 
	NOT prgLinuxCommand.METH_IsDockerBTActive()
	AND prgLinuxCommand.METH_IsDockerDoosanActive()
	AND prgEIPMapping.METH_IsDoosanServoOn(DoosanState := prgEIPMapping.DoosanState)
;
                        
END_METHOD

METHOD METH_WaitingForCommands : BOOL
                          METH_WaitingForCommands := eStep = step_enum_t.Dormant;
                        
END_METHOD

METHOD METH_ARunWasGiven : BOOL
                          METH_ARunWasGiven := xARunWasGiven;
                        
END_METHOD

METHOD METH_DetectInitializing : BOOL
                          METH_DetectInitializing := iStepInit > 0;
                        
END_METHOD

METHOD METH_DetectVision : BOOL
  VAR_INPUT
    eProcStat : process_code_enum_t;
  END_VAR
                          METH_DetectVision := FALSE; //eProcStat = process_code_enum_t.pcode_Vision;
                        
END_METHOD
END_PROGRAM

PROGRAM prgApplica
  VAR
    xTB_WriteMachineStatus : BOOL;
    xTB_RaiseEvent : BOOL;
    eTestMachineState : machine_state_enum_t;
    TON_SimulateProdOK : Standard.TON;
    xSimulateProdOK : BOOL;
    tSimulateProdOK : TIME := TIME#10s0ms;
    TON_SimulateProdNotOK : Standard.TON;
    xSimulateProdNotOK : BOOL;
    tSimulateProdNotOK : TIME := TIME#30s0ms;
    xTB_ResetOverallCounters : BOOL;
    xTB_ResetSessionCounters : BOOL;
    xInit : BOOL := TRUE;
    pRtcRes : SysTimeRtc.RTS_IEC_RESULT;
    dwRtcTime : DWORD;
    dtSessionStart : DT;
    dtRtcTime : DT;
    dwPrevRtcTime : DWORD;
    dwDiff : DWORD;
    xIsUpTime : BOOL;
    xAllowCounters : BOOL;
    liDiff : LINT;
    dwMachineStateFontColor : DWORD;
    dwMachineErrorFontColor : DWORD;
    xwCurrentRtcTime : __XWORD;  (* eProposedMachineState: machine_state_enum_t; eProposedMachineError: machine_error_enum_t; *)
    pResultGetTime : SysTimeRtc.RTS_IEC_RESULT;
    uliNsTickTime : SysTimeCore.SYSTIME;
    udiResNs : UDINT;
    uliSeed : ULINT;
    eGenRndError : SysDesignUUID.ERROR;
    bMyRndByte : BYTE;
    iMinDepth : INT := 15;
    iMaxDepth : INT := 25;
    iDepthSpan : INT := 10;
    TON_ChangeDepth : TON;
    tChangeDepth : TIME := TIME#30s0ms;
    aePiecesStates : ARRAY[0..c_iMaxIndDepth] OF piece_state_enum_t;
    xAutoChangeDepthFlag : BOOL;  (* xPausedWhileRunning: BOOL; *)
  END_VAR
  VAR CONSTANT
    c_Red : DWORD := 16#FFFF0000;
    c_Green : DWORD := 16#FF99FFCC;
    c_Blue : DWORD := 16#FF0000FF;
    c_White : DWORD := 16#FFFFFFFF;
    c_iMaxDepth : INT := 25;
    c_iMaxIndDepth : INT := (c_iMaxDepth - 1);
  END_VAR

                    // initialization
// RTC time count (UTC)
dwRtcTime := SysTimeRtc.SysTimeRtcGet(pResult := pRtcRes);
dtRtcTime := DWORD_TO_DT(dwRtcTime);
IF xInit THEN
	xInit := FALSE;
	dtSessionStart := dtRtcTime;
	GVL_Applica.g_SessionCounters.dtUTCStartCounting := dtSessionStart;
END_IF
(*-------------------------------------------------------------*)
// impose machine state
IF xTB_WriteMachineStatus THEN
	xTB_WriteMachineStatus := FALSE;
	GVL_Applica.g_MachineMESInterface.Machine.eState := eTestMachineState;
END_IF
(*-------------------------------------------------------------*)
// SIMULATE production

// PIECE OK
TON_SimulateProdOK(IN := xSimulateProdOK, PT := tSimulateProdOK);
IF TON_SimulateProdOK.Q THEN
	TON_SimulateProdOK(IN := FALSE);
	METH_IncreaseCounter_PieceOK();
END_IF

// PIECE NOT OK
TON_SimulateProdNotOK(IN := xSimulateProdNotOK, PT := tSimulateProdNotOK);
IF TON_SimulateProdNotOK.Q THEN
	TON_SimulateProdNotOK(IN := FALSE);
	METH_IncreaseCounter_PieceNotOK();
END_IF
(*-------------------------------------------------------------*)
// Reset counters
IF xTB_ResetOverallCounters THEN
	xTB_ResetOverallCounters := FALSE;
	METH_OverallCountersReset();
	METH_SessionCountersReset();
END_IF

IF xTB_ResetSessionCounters THEN
	xTB_ResetSessionCounters := FALSE;
	METH_SessionCountersReset();
END_IF
(*-------------------------------------------------------------*)
// increase time counter
// at each cycle, sum the difference
IF dwPrevRtcTime > 0 AND xAllowCounters THEN
	liDiff := DWORD_TO_LINT(dwRtcTime) - DWORD_TO_LINT(dwPrevRtcTime); // time difference from last execution
	IF liDiff > 0 THEN
		dwDiff := LINT_TO_DWORD(liDiff);
		xIsUpTime := TRUE;
		CASE GVL_Applica.g_MachineMESInterface.Machine.eState OF
			machine_state_enum_t.MachineUnknownState:
				//
			(*-------------------------------------------------------*)
			machine_state_enum_t.MachineReady:
				METH_IncreaseTimeCounter_Ready();
			(*-------------------------------------------------------*)
			machine_state_enum_t.MachineRunning:
				METH_IncreaseTimeCounter_Running();
			(*-------------------------------------------------------*)
			machine_state_enum_t.MachineError:
				METH_IncreaseTimeCounter_Error();
			(*-------------------------------------------------------*)
			ELSE
				//
		END_CASE
		IF xIsUpTime THEN
			METH_IncreaseTimeCounter_UpTime();
		END_IF
	END_IF
ELSE
	IF dwRtcTime > 0 THEN
		xAllowCounters := TRUE;
	END_IF
END_IF
dwPrevRtcTime := dwRtcTime;
(*-------------------------------------------------------------*)
// Pass counters to Machine interface
GVL_Applica.g_MachineMESInterface.Counters.LastSession := GVL_Applica.g_SessionCounters;
GVL_Applica.g_MachineMESInterface.Counters.Overall := PersVars.g_OverallCounters;


(*-------------------------------------------------------------*)
// IF xTB_RaiseEvent THEN
// 	xTB_RaiseEvent := FALSE;
// 	AlarmManager.AlarmGlobals.g_AlarmHandler.RaiseEvent(
// 		Alm_AlarmConfiguration_Alarmgroup_IDs.ID_ApplicationEvent, Alm_ApplicationEvent_Alarm_IDs.ID_0
// 	);
// END_IF

CASE GVL_Applica.g_MachineMESInterface.Machine.eState OF
	machine_state_enum_t.MachineSafetyStop, machine_state_enum_t.MachineSafeguardStop, machine_state_enum_t.MachineError:
		dwMachineStateFontColor := c_Red;
	(*---------------------------------------------------------*)
	machine_state_enum_t.MachineRunning:
		dwMachineStateFontColor := c_Green;
	(*---------------------------------------------------------*)
	ELSE
		dwMachineStateFontColor := c_White;
END_CASE

CASE  GVL_Applica.g_MachineMESInterface.Machine.eError OF
	machine_error_enum_t.NO_ERROR:
		dwMachineErrorFontColor := c_White;
	(*---------------------------------------------------------*)
	ELSE
		dwMachineErrorFontColor := c_Red;
END_CASE
(*-------------------------------------------------------------*)
(*-------------------------------------------------------------*)
// DEPTH for statistic
TON_ChangeDepth(IN := GVL.g_xRUNNING AND xAutoChangeDepthFlag, PT := tChangeDepth);
iMaxDepth := c_iMaxDepth;
IF TON_ChangeDepth.Q THEN
	TON_ChangeDepth(IN := FALSE);
	xwCurrentRtcTime := SysTimeRtcGet(pResultGetTime);
	udiResNs := SysTimeGetNs(pUsTime := uliNsTickTime);
	uliSeed := __XWORD_TO_ULINT(xwCurrentRtcTime) + uliNsTickTime;
	eGenRndError := SysDesignUUID.FUN_GenerateRnd_x64(uliSeed := uliSeed, xInit := TRUE, bOutput => bMyRndByte); // between 0 and 255
	
	GVL_Applica.g_iDepth := LIMIT(iMinDepth, (BYTE_TO_INT(bMyRndByte) MOD iDepthSpan) + iMinDepth, iMaxDepth); // random depth
ELSE
	// fixed depth
	iMaxDepth := __UXINT_TO_INT(XSIZEOF(aePiecesStates)/XSIZEOF(aePiecesStates[0]));
	GVL_Applica.g_iDepth := LIMIT(iMinDepth, GVL_Applica.g_iDepth, iMaxDepth); // limit depth
END_IF



                  

METHOD METH_IncreaseCounter_PieceOK
                          GVL_Applica.g_SessionCounters.udiPiecesOK_Counter := GVL_Applica.g_SessionCounters.udiPiecesOK_Counter + 1;
PersVars.g_OverallCounters.udiPiecesOK_Counter := PersVars.g_OverallCounters.udiPiecesOK_Counter + 1;
                        
END_METHOD

METHOD METH_IncreaseCounter_PieceNotOK
                          GVL_Applica.g_SessionCounters.udiPiecesNotOK_Counter := GVL_Applica.g_SessionCounters.udiPiecesNotOK_Counter + 1;
PersVars.g_OverallCounters.udiPiecesNotOK_Counter := PersVars.g_OverallCounters.udiPiecesNotOK_Counter + 1;
                        
END_METHOD

METHOD METH_OverallCountersReset
                          SysMem.SysMemSet(
	pDest := ADR(PersVars.g_OverallCounters),
	udiCount := XSIZEOF(PersVars.g_OverallCounters),
	udiValue := 0
);

PersVars.g_OverallCounters.dtUTCStartCounting := dtRtcTime;
                        
END_METHOD

METHOD METH_SessionCountersReset
                          SysMem.SysMemSet(
	pDest := ADR(GVL_Applica.g_SessionCounters),
	udiCount := XSIZEOF(GVL_Applica.g_SessionCounters),
	udiValue := 0
);

GVL_Applica.g_SessionCounters.dtUTCStartCounting := dtRtcTime;
                        
END_METHOD

METHOD METH_IncreaseTimeCounter_UpTime
                          GVL_Applica.g_SessionCounters.dwUpTime := GVL_Applica.g_SessionCounters.dwUpTime + dwDiff;
PersVars.g_OverallCounters.dwUpTime := PersVars.g_OverallCounters.dwUpTime + dwDiff;
                        
END_METHOD

METHOD METH_IncreaseTimeCounter_Ready
                          GVL_Applica.g_SessionCounters.dwReadyTime := GVL_Applica.g_SessionCounters.dwReadyTime + dwDiff;
PersVars.g_OverallCounters.dwReadyTime := PersVars.g_OverallCounters.dwReadyTime + dwDiff;
                        
END_METHOD

METHOD METH_IncreaseTimeCounter_Running
                          GVL_Applica.g_SessionCounters.dwRunningTime := GVL_Applica.g_SessionCounters.dwRunningTime + dwDiff;
PersVars.g_OverallCounters.dwRunningTime := PersVars.g_OverallCounters.dwRunningTime + dwDiff;
                        
END_METHOD

METHOD METH_IncreaseTimeCounter_Error
                          GVL_Applica.g_SessionCounters.dwErrorTime := GVL_Applica.g_SessionCounters.dwErrorTime + dwDiff;
PersVars.g_OverallCounters.dwErrorTime := PersVars.g_OverallCounters.dwErrorTime + dwDiff;
                        
END_METHOD

METHOD METH_AnalyzeLatestResults : INT
  VAR_INPUT
    iDepth : INT;
  END_VAR
  VAR_OUTPUT
    xFlipNext : BOOL;
    lrCurrentNotOKRatio : LREAL;
  END_VAR
  VAR
    iMaxInd : INT;
    xParsingOK : BOOL;
    iInd : INT;
    iCounterOK : INT;
    iCounterNOT_OK : INT;
    iTotal : INT;
    lrPercentageNOT_OK : LREAL;
    lrMinErr : LREAL := 0.15;
    lrMaxErr : LREAL := 0.25;
    udiResRndNs : UDINT;
    xRandomCond : BOOL;
    uliLocalNsTickTime : SysTimeCore.SYSTIME;
  END_VAR
                          xParsingOK := iDepth > 0;
IF xParsingOK THEN
	iMaxInd := iDepth - 1;
	FOR iInd := 0 TO iMaxInd DO // counters all over the history
		IF aePiecesStates[iInd] = piece_state_enum_t.PieceOK THEN
			iCounterOK := iCounterOK + 1;
		ELSIF aePiecesStates[iInd] = piece_state_enum_t.PieceNotOK THEN
			iCounterNOT_OK := iCounterNOT_OK + 1;
		END_IF
	END_FOR
	iTotal := iCounterOK + iCounterNOT_OK;
	IF iTotal > 0 THEN
		lrPercentageNOT_OK := INT_TO_LREAL(iCounterNOT_OK) / INT_TO_LREAL(iTotal);
		IF lrPercentageNOT_OK < lrMinErr THEN // low percentage -> introduce error
			xFlipNext := TRUE;
		ELSIF lrPercentageNOT_OK > lrMaxErr THEN // high percentage -> no error
			xFlipNext := FALSE;
		ELSE // in the middle
			udiResRndNs := SysTimeGetNs(pUsTime := uliLocalNsTickTime);
			xRandomCond := (uliLocalNsTickTime MOD 3) = 0;
			xFlipNext := xRandomCond;
		END_IF
	END_IF
END_IF

lrCurrentNotOKRatio := lrPercentageNOT_OK;
METH_AnalyzeLatestResults := iTotal;

                        
END_METHOD

METHOD METH_InsertIntoHistory
  VAR_INPUT
    xIsOk : BOOL;
  END_VAR
  VAR_IN_OUT
    iInd : INT;
  END_VAR
  VAR
    iHistoryArrDim : INT;
    iMaxVal : INT;
  END_VAR
                          IF xIsOk THEN
	aePiecesStates[iInd] := piece_state_enum_t.PieceOK;
ELSE
	aePiecesStates[iInd] := piece_state_enum_t.PieceNotOK;
END_IF

iHistoryArrDim := __UXINT_TO_INT(XSIZEOF(aePiecesStates)/XSIZEOF(aePiecesStates[0]));
iMaxVal := MIN(GVL_Applica.g_iDepth, iHistoryArrDim);

iInd := (iInd + 1) MOD iMaxVal;
                        
END_METHOD
END_PROGRAM

PROGRAM prgLight
  VAR
    LightManager : FB_LightManager;
    CTRL_Light : SysDesignBasic.SysD_basic_ctrl_struct_t := (xExecute := TRUE);
    eLightError : SysDesignBasic.LIGHT_ERROR;
    eLightStep : SysDesignBasic.Steps_Light_t;
  END_VAR

                    LightManager(
	xEnable := CTRL_Light.xExecute,
	xBusy => CTRL_Light.xProcessing,
	xError => CTRL_Light.xFailure,
	
	pxGreen := ADR(GVL.g_LightTower.xGreen),
	pxYellow := ADR(GVL.g_LightTower.xYellow),
	pxRed := ADR(GVL.g_LightTower.xRed),
	
	eErrorID => eLightError,
	eCurrentStep => eLightStep,
	sLightMessage => CTRL_Light.sStatusMessage
);
                  
END_PROGRAM

FUNCTION_BLOCK FB_LightManager EXTENDS SysDesignBasic.FB_LightManager_TPL

                    SUPER^();
                  

(* {warning 'Add method implementation '} *)
METHOD METH_SetLightStep : SysDesignBasic.Steps_Light_t
  VAR_OUTPUT
    sMessage : STRING(255);
  END_VAR
  VAR
    eRes : SysDesignBasic.Steps_Light_t := SysDesignBasic.Steps_Light_t.Light_EasterEag;
    xProblemSpecified : BOOL := TRUE;
  END_VAR
                          IF NOT GVL.g_xSafetyOK THEN
	eRes := SysDesignBasic.Steps_Light_t.Light_EmergencyStop;
ELSE
	IF NOT GVL.g_xSafeguardOK THEN
		eRes := SysDesignBasic.Steps_Light_t.Light_StoppedOperatorRequest;
	ELSE
		IF GVL_Applica.g_MachineMESInterface.Machine.eState = machine_state_enum_t.MachineError THEN
			eRes := SysDesignBasic.Steps_Light_t.Light_StoppedOperatorRequest;
		ELSIF GVL_Applica.g_MachineMESInterface.Machine.eState = machine_state_enum_t.MachineToInitialize THEN
			eRes := SysDesignBasic.Steps_Light_t.Light_MachineWorkOperatorRequest;
		ELSIF GVL_Applica.g_MachineMESInterface.Machine.eState = machine_state_enum_t.MachineReady THEN
			eRes := SysDesignBasic.Steps_Light_t.Light_ReadyButNotWork;		ELSE
			IF GVL_Applica.g_MachineMESInterface.Machine.eState = machine_state_enum_t.MachinePaused THEN
				eRes := SysDesignBasic.Steps_Light_t.Light_ReadyButNotWork;
			ELSIF GVL_Applica.g_MachineMESInterface.Machine.eState = machine_state_enum_t.MachineOperatorInteraction THEN
				eRes := SysDesignBasic.Steps_Light_t.Light_MachineWorkOperatorRequest;
			ELSIF GVL_Applica.g_MachineMESInterface.Machine.eState = machine_state_enum_t.MachineWarning THEN
				eRes := SysDesignBasic.Steps_Light_t.Light_MachineWorkOperatorRequest;
			ELSE
IF GVL_Applica.g_MachineMESInterface.Machine.eState = machine_state_enum_t.MachineRunning THEN
					eRes := SysDesignBasic.Steps_Light_t.Light_MachineWork;
				ELSE
					// default pattern
				END_IF
			END_IF
		END_IF
	END_IF
END_IF

METH_SetLightStep := eRes;
                        
END_METHOD

(* {warning 'Add method implementation '} *)
METHOD METH_ParseCustomInputs : BOOL
                          METH_ParseCustomInputs := TRUE;
                        
END_METHOD
END_FUNCTION_BLOCK

PROGRAM Reboot_Application
  VAR
    R_TRIGReset : R_TRIG;
    ResetPLC : BOOL;
    pApp : POINTER TO Application;
    xSavedSafeguardPosOK : BOOL;
    xReqRebootPLC : BOOL;
  END_VAR

                    
R_TRIGReset(CLK:=ResetPLC AND NOT GVL_HMI.DisableReboot);
IF R_TRIGReset.Q THEN
	xReqRebootPLC:=TRUE;
END_IF

IF xReqRebootPLC  THEN
	SysDesignBasic.BASIC_ResetApplication();
END_IF
                  
END_PROGRAM

FUNCTION Restart : DWORD
  VAR_IN_OUT
    EventPrm : CmpApp.EVTPARAM_CmpAppReset;
  END_VAR

                    Restart := SysDesignBasic.BASIC_AutostartApplication(EVTPARAM_EventPrm := EventPrm);
                  
END_FUNCTION

FUNCTION FUN_ROSPose2Quat : SMC_Quat
  VAR_INPUT
    Ori : ROS_orientation_struct_t;
  END_VAR
  VAR
    Res : SMC_Quat;
  END_VAR

                    Res.dR := Ori.w;
Res.dI := Ori.x;
Res.dJ := Ori.y;
Res.dK := Ori.z;

FUN_ROSPose2Quat := Res;
                  
END_FUNCTION

PROGRAM prg_HMI_MainFrame
  VAR
    iSelectionMainFrameView : INT;
    BlinkSyncSlow : Util.BLINK;
    BlinkSyncFast : Util.BLINK;
    tSlowLow : TIME := TIME#1s0ms;
    tSlowHigh : TIME := TIME#1s0ms;
    tFastLow : TIME := TIME#500ms;
    tFastHigh : TIME := TIME#500ms;
    xOutSlow : BOOL;
    xOutFast : BOOL;
  END_VAR

                    ACT_BlinkingSync();
                  

ACTION ACT_BlinkingSync:
                        BlinkSyncSlow(
	ENABLE := TRUE,
	TIMELOW := tSlowLow,
	TIMEHIGH := tSlowHigh,
	
	OUT => xOutSlow
);

BlinkSyncFast(
	ENABLE := TRUE,
	TIMELOW := tFastLow,
	TIMEHIGH := tFastHigh,
	
	OUT => xOutFast
);
                      
END_ACTION

METHOD Init
  VAR
    stSrc : STRING;
    stDest : STRING;
  END_VAR
                          
// stSrc := '$$PlcLogic$$/Application/video.htm';
// stDest := '$$PlcLogic$$/$$visu$$/video.htm';
// SysFile.SysFileCopy(stDest, stSrc, 0);

// stSrc := '$$PlcLogic$$/Application/video.mp4';
// stDest := '$$PlcLogic$$/$$visu$$/video.mp4';
// SysFile.SysFileCopy(stDest, stSrc, 0);
stSrc := '$$PlcLogic$$/Application/21UT01.pdf';
stDest := '$$PlcLogic$$/$$visu$$/21UT01.pdf';
SysFile.SysFileCopy(stDest, stSrc, 0);
VisuElems.VisuElemBase.g_VisuEventManager.SetMouseEventHandler(PLC_PRG.evHandler);
                        
END_METHOD

METHOD METH_GetBlinkSync_Slow : BOOL
                          METH_GetBlinkSync_Slow := xOutSlow;
                        
END_METHOD

METHOD METH_GetBlinkSync_Fast : BOOL
                          METH_GetBlinkSync_Fast := xOutFast;
                        
END_METHOD
END_PROGRAM

PROGRAM prgLinuxCommand_OLD
  VAR
    xTB_LinuxCommandTest : BOOL;
    xTB_NodeList : BOOL;
    diProcessExecuteResult : DINT;
    RTS_Result : SysProcess.RTS_IEC_RESULT;
    sCommand : STRING(255) := 'sudo pwd';
    sStdOutBuffer : STRING(1000);
    udiSizeStdOutBuffer : UDINT;
    iCounterFailure : INT;
    iCounterSuccess : INT;
    sLastStdOutResult : STRING(1000);
    sErrorMessage : STRING;
    xwCopySize : __XWORD;
    sPythonFile_Echo : STRING := 'echo.py';
    sPythonCommand_Echo : STRING(255) := 'CONCAT(c_sPythonExecute, sPythonFile_Echo)';
    sDestFullPath_Echo : STRING(255);
    sSourceFullPath_Echo : STRING(255);
    sBashFile_DockerActivate : STRING := 'launch_docker.sh';
    sBashCommand_DockerActivate : STRING(255) := 'CONCAT(c_sBashExecute, sBashFile_DockerActivate)';
    sDestFullPath_DockerActivate : STRING(255);
    sSourceFullPath_DockerActivate : STRING(255);
    sBashFile_RobinActivate : STRING := 'launch_remote_robin.sh';
    sBashCommand_RobinActivate : STRING(255) := 'CONCAT(c_sBashExecute, sBashFile_RobinActivate)';
    sDestFullPath_RobinActivate : STRING(255);
    sSourceFullPath_RobinActivate : STRING(255);
    xTB_ActivateDocker : BOOL;
    xTB_ActivateRobin : BOOL;
    sTestCommand : STRING(255) := 'sudo roscore';
    xTB_ShutdownMiniPC : BOOL;
    xDIS_Command : BOOL;
    xTB_RebootMiniPC : BOOL;
    xTB_StartDocker : BOOL;
    xTB_KillBehaviorTree : BOOL;
    xTB_StartBehaviorTree : BOOL;
    xTB_StopDocker : BOOL;
    xTB_ListDockers : BOOL;
    xListContainers : BOOL;
    sContainersAlive : STRING(255);
    xTB_KillBoxDetection : BOOL;
    xTB_StartBoxDetection : BOOL;
    xTB_ReadFile : BOOL;
    RTS_FileCloseResult : SysTypes.RTS_IEC_RESULT;
    xListNodes : BOOL;
    sNodesAlive : STRING(255);
    TON_NodeList : TON;
    xTB_NodeListStartNode : BOOL;
    tTimeStart : TIME := TIME#3s0ms;
    TON_NodeListPolling : TON;
    xIsDockerStarted : BOOL;
    tPollingNodes : TIME := TIME#10s0ms;
    xTB_StartDoosanControl : BOOL;
    xTB_KillDoosanControl : BOOL;
    xTB_StartDoosanMover : BOOL;
    xTB_KillDoosanMover : BOOL;
    xIsDoosanControlStarted : BOOL;
    xIsDoosanMoverStarted : BOOL;
    xIsBoxRecognitionStarted : BOOL;
    xIsBehaviorStarted : BOOL;
    tPollingDocker : TIME := TIME#30s0ms;
    TON_DockerListPolling : TON;
    iStepStartAll : INT;
    xTB_StartAllNodes : BOOL;
    xNodeStartRequested : BOOL;
    xTB_StopAllNodes : BOOL;
    xAllNodesDown : BOOL;
    xAllNodesAreUp : BOOL;
    xTB_START : BOOL;
    xTB_STOP : BOOL;
    xTB_RECOVERY_TOOL_EMPTY : BOOL;
    xEnableListing : BOOL;
    xTB_RECOVERY_TOOL_BUNDLE : BOOL;
  END_VAR
  VAR CONSTANT
    c_sDestPath : STRING := '/var/opt/codesys/';
    c_sSourcePath : STRING := '/var/opt/codesys/PlcLogic/Application/';
    c_sPythonExecute : STRING := 'sudo python ';
    c_sBashExecute : STRING := './';
    c_sDockerName : STRING := 'philip_production';  (* philip_development //philip_devel-v2 //philip_development *)
    c_sDockerActivateFile : STRING := 'launch_docker.sh';
  END_VAR

                    (*=======================================================*)
// MINI PC
IF xTB_ShutdownMiniPC OR GVL.g_xShutdownMiniPC THEN
	GVL.g_xShutdownMiniPC := FALSE;
	xTB_ShutdownMiniPC := FALSE;
	sTestCommand := 'sudo shutdown -h now';
	xTB_LinuxCommandTest := TRUE;
END_IF
IF xTB_RebootMiniPC OR GVL.g_xRebootMiniPC THEN
	GVL.g_xRebootMiniPC := FALSE;
	xTB_RebootMiniPC := FALSE;
	sTestCommand := 'sudo reboot';
	xTB_LinuxCommandTest := TRUE;
END_IF

(*--------------------------------*)
// DOCKER
TON_DockerListPolling(IN := xEnableListing, PT := tPollingDocker);
IF TON_DockerListPolling.Q THEN
	TON_DockerListPolling(IN := FALSE);
	xTB_ListDockers := TRUE;
END_IF
IF xTB_ListDockers OR GVL.g_xListDockers THEN
	GVL.g_xListDockers := FALSE;
	xTB_ListDockers := FALSE;
	sTestCommand := 'docker container ls';
	xTB_LinuxCommandTest := TRUE;
	xListContainers := TRUE;
END_IF

xIsDockerStarted := FIND(sContainersAlive, c_sDockerName) > 0;
TON_NodeListPolling(IN := xIsDockerStarted AND xEnableListing, PT := tPollingNodes);
IF TON_NodeListPolling.Q THEN
	TON_NodeListPolling(IN := FALSE);
	xTB_NodeList := TRUE;
END_IF
(*===============================================*)
// LIST
IF xTB_NodeList THEN
	xTB_NodeList := FALSE;
// 	sTestCommand := './launch_docker.sh';
	sTestCommand := '';
// 	sTestCommand := 'docker exec ';
// 	sTestCommand := CONCAT(sTestCommand, c_sDockerName);
// 	sTestCommand := CONCAT(sTestCommand, ' bash -c $'source devel/setup.bash; rosnode list$'');
	sTestCommand := 'bash -c $'source /opt/ros/noetic/setup.bash; rosnode list$'';
	xTB_LinuxCommandTest := TRUE;
	xListNodes := TRUE;
END_IF
(*--------------------------------*)
// 20/09/2022 COMPREHENSIVE COMMANDS
IF xTB_START OR GVL.g_xNODES_START THEN
	xTB_START := FALSE;
	GVL.g_xNODES_START := FALSE;
	sTestCommand := '';
	IF GVL.g_xLocalTestMachine THEN
		sTestCommand := 'docker compose -f /home/nicola/ros/exhibition_ws/src/mecspe-exhibition/docker-compose.devel.yml up -d';
	ELSE
		sTestCommand := 'bash /home/sysdesign/philip.sh start';
	END_IF
	xTB_LinuxCommandTest := TRUE;
END_IF

IF xTB_STOP OR GVL.g_xNODES_STOP THEN
	xTB_STOP := FALSE;
	GVL.g_xNODES_STOP := FALSE;
	IF GVL.g_xLocalTestMachine THEN
		sTestCommand := 'docker compose -f /home/nicola/ros/exhibition_ws/src/mecspe-exhibition/docker-compose.devel.yml down';
	ELSE
		sTestCommand := 'bash /home/sysdesign/philip.sh stop';
	END_IF
	xTB_LinuxCommandTest := TRUE;
END_IF

// IF xTB_RECOVERY_TOOL_EMPTY OR GVL.g_xRECOVERY_EMPTY THEN
// 	xTB_RECOVERY_TOOL_EMPTY := FALSE;
// 	GVL.g_xRECOVERY_EMPTY := FALSE;
// 	sTestCommand := 'bash /home/sysdesign/philip.sh recover --tool PM01_EMPTY_SW';
// 	xTB_LinuxCommandTest := TRUE;
// END_IF
// 
// IF xTB_RECOVERY_TOOL_BUNDLE OR GVL.g_xRECOVERY_BUNDLE THEN
// 	xTB_RECOVERY_TOOL_BUNDLE := FALSE;
// 	GVL.g_xRECOVERY_BUNDLE := FALSE;
// 	sTestCommand := 'bash /home/sysdesign/philip.sh recover --tool PM01_BUNDLE_SW';
// 	xTB_LinuxCommandTest := TRUE;
// END_IF
(*--------------------------------*)

(*--------------------------------*)
// flags
xIsDoosanControlStarted := FIND(sNodesAlive, 'dsr01h2017') > 0;
xIsDoosanMoverStarted := FIND(sNodesAlive, 'doosan_mover') > 0;
xIsBoxRecognitionStarted := FIND(sNodesAlive, 'box_recognition') > 0;
xIsBehaviorStarted := FIND(sNodesAlive, 'behavior_tree') > 0;
(*--------------------------------*)
xDIS_Command := FALSE;
IF xTB_LinuxCommandTest THEN
	xTB_LinuxCommandTest := FALSE;
	
	sCommand := sTestCommand;
// 	sCommand := sPythonCommand_Echo;
	
	sErrorMessage := '';
	udiSizeStdOutBuffer := TO_UDINT(XSIZEOF(sStdOutBuffer));
	SysMem.SysMemSet(pDest := ADR(sStdOutBuffer), udiCount := XSIZEOF(sStdOutBuffer), udiValue := 0);
	
	diProcessExecuteResult := SysProcess.SysProcessExecuteCommand2(
		pszCommand := sCommand,
		pResult := ADR(RTS_Result),
		pszStdOut := sStdOutBuffer,
		udiStdOutLen := udiSizeStdOutBuffer
	);
	
	IF RTS_Result = CmpErrors.Errors.ERR_OK THEN
		iCounterSuccess := (iCounterSuccess + 1) MOD 16#7FFF;
		IF diProcessExecuteResult > 0 THEN // there is something to read
			sLastStdOutResult := sStdOutBuffer;
		END_IF
		IF xListContainers THEN
			xListContainers := FALSE;
			sContainersAlive := sStdOutBuffer;
		END_IF
		IF xListNodes THEN
			xListNodes := FALSE;
			sNodesAlive := sStdOutBuffer;
		END_IF
	ELSE
		sErrorMessage := METH_GetErrorMessage(udiResult := RTS_Result);
		iCounterFailure := (iCounterFailure + 1) MOD 16#7FFF;
		IF xListNodes THEN
			xListNodes := FALSE;
			sNodesAlive := '';
		END_IF
	END_IF
END_IF

                  

METHOD METH_GetErrorMessage : STRING(255)
  VAR_INPUT
    udiResult : SysProcess.RTS_IEC_RESULT;
  END_VAR
  VAR
    sRes : STRING(255);
  END_VAR
                          CASE udiResult OF
	CmpErrors.Errors.ERR_PARAMETER:
		sRes := 'Some null input parameter';
	CmpErrors.Errors.ERR_NO_ACCESS_RIGHTS:
		sRes := 'Not allowed';
	CmpErrors.Errors.ERR_FAILED:
		sRes := 'Internal error';
	ELSE
		sRes := 'Error';
END_CASE

METH_GetErrorMessage := sRes;
                        
END_METHOD
END_PROGRAM

PROGRAM prg_Hmi_Home
  VAR
    sDescriptionBar : STRING(255) := '23KR01 - vX.X.X';  (* - - *)
    sStatusMessage : STRING(255);
    xDIS_Play : BOOL;
    xDIS_Pause : BOOL;
    xDIS_Stop : BOOL;
    xDIS_Reset : BOOL;
    xDIS_DoosanButton : BOOL;
    xTB_TurnDoosanOFF : BOOL;
    xTB_TurnDoosanON : BOOL;
    xTurningON : BOOL;
    xTurningOFF : BOOL;
    TON_ON : TON;
    TON_OFF : TON;
    tTurnOn : TIME := TIME#1s0ms;
    tTurnOff : TIME := TIME#20s0ms;
    xTB_Retry : BOOL;
    xDIS_Retry : BOOL;
    xIsBTStateTrustworthy : BOOL;
    xDIS_IsBTStateTrustworthy : BOOL;
    dwMachineStateColor : DWORD;
    xErrorToRetry : BOOL;
  END_VAR

                    sDescriptionBar := 'DEMO PallCUBE - v1.0.0'; //24/10/2022

IF GVL_HMI.xPlay THEN
	GVL_HMI.xPlay := FALSE;
	GVL.g_xPLAY := TRUE;
END_IF

GVL.g_xPAUSE := GVL_HMI.xPause;

IF GVL_HMI.xReload THEN
	GVL_HMI.xReload := FALSE;
	GVL.g_xRESET := TRUE;
END_IF

IF GVL_HMI.xStop THEN
	GVL_HMI.xStop := FALSE;
	GVL_HMI.g_xIsStoppedByUser := TRUE;
	GVL.g_xSTOP := TRUE;
END_IF
(**)

xDIS_DoosanButton := xTurningON OR xTurningOFF; //12/01/2023: FALSE

IF xTB_TurnDoosanON THEN
	xTB_TurnDoosanON := FALSE;
	xTurningON := TRUE;
	GVL.g_xDoosanButton := TRUE;
END_IF

TON_ON(IN := xTurningON, PT := tTurnOn);
IF TON_ON.Q THEN
	TON_ON(IN := FALSE);
	xTurningON := FALSE;
	GVL.g_xDoosanButton := FALSE;
END_IF

IF xTB_TurnDoosanOFF THEN
	xTB_TurnDoosanOFF := FALSE;
	xTurningOFF := TRUE;
	GVL.g_xDoosanButton := TRUE;
END_IF
TON_OFF(IN := xTurningOFF, PT := tTurnOff);
IF TON_OFF.Q THEN
	TON_OFF(IN := FALSE);
	xTurningOFF := FALSE;
	GVL.g_xDoosanButton := FALSE;
END_IF

(**)


xDIS_Play := 
	GVL_Applica.g_MachineMESInterface.Machine.eState <> machine_state_enum_t.MachineReady
	OR GVL.g_xRUNNING
;

xDIS_Pause := NOT GVL.g_xRUNNING OR GVL_Hmi.g_xIsStoppedByUser;
xDIS_Stop := NOT GVL.g_xRUNNING OR GVL_Hmi.g_xIsStoppedByUser;
xDIS_Reset := 
	GVL_Applica.g_MachineMESInterface.Machine.eState <> machine_state_enum_t.MachineError
	OR prgLinuxCommand.METH_IsDockerBTActive()
;
(**)
xErrorToRetry := 
	GVL.g_xRUNNING 
	AND prgROS.xThereIsROSError_01 
	AND NOT TO_BOOL(prgROS.ROSInterface_01.Codesys2ROS.Published.run)
;
xDIS_Retry := NOT xErrorToRetry
	OR prgMain.METH_WaitingForCommands()
;
IF xTB_Retry THEN
	xTB_Retry := FALSE;
	prgROS.METH_SetRun_01(xValue := TRUE);
END_IF

(*---------------------------------------*)
xIsBTStateTrustworthy :=
	prgLinuxCommand.METH_IsDockerBTActive()
	AND prgMain.METH_ARunWasGiven()
;

xDIS_IsBTStateTrustworthy := NOT xIsBTStateTrustworthy;

(*---------------------------------------------------*)
                  

METHOD METH_AskForDoosanOff
                          xTB_TurnDoosanOFF := TRUE;
                        
END_METHOD

METHOD METH_AskForDoosanOn
                          xTB_TurnDoosanON := TRUE;
                        
END_METHOD
END_PROGRAM

PROGRAM prg_HMI_MiniPCMenu
  VAR
    sDescriptionBar : STRING(255) := 'Stato menu CubeOS:';
    sStatusMessage : STRING(255);
    dwFleetErrorColor : DWORD;
  END_VAR

                    // IF visuElems.CURRENTLANGUAGE = 'it' THEN
// 	sDescriptionBar := 'Menù MiniPC:';
// ELSE
// 	sDescriptionBar := 'MiniPC menu:';
// END_IF

// sStatusMessage := GVL.g_PM_HMI_StatusMessages.sMiniPCMenu;


